(* Logix 5000 project; controller AMANA_DC_PLANT_01 vendor 1 type 14 code 164 rev 31.12; software revision 31.02; part 2 of 9 *)

TYPE Keyence_2_Barcode :
STRUCT
   Trigger_Timer : TIMER;
   Barcode_SRTrigger : BOOL;
   Barcode_ReadIsSuccess : BOOL;
   Barcode_Raw : STRING;
   Barcode_Comma_Position : INT;
   Barcode_1_Length : INT;
   Barcode_2_Length : INT;
   Barcode_2_Start : INT;
   PlaceHolder_ConveyorRunning : BOOL;
   Barcode_1_String : STRING;
   Barcode_2_String : STRING;
   Scanner_Name : STRING;
   Barcode_SRReaderReady : BOOL;
   OneShot : BOOL;
END_STRUCT
END_TYPE

TYPE STRING_12 :
STRUCT
   LEN : DINT;
   DATA : SINT[12];
END_STRUCT
END_TYPE

TYPE STRING_16 :
STRUCT
   LEN : DINT;
   DATA : SINT[16];
END_STRUCT
END_TYPE

TYPE STRING_24 :
STRUCT
   LEN : DINT;
   DATA : SINT[24];
END_STRUCT
END_TYPE

TYPE STRING_4 :
STRUCT
   LEN : DINT;
   DATA : SINT[4];
END_STRUCT
END_TYPE

TYPE STRING_40 :
STRUCT
   LEN : DINT;
   DATA : SINT[40];
END_STRUCT
END_TYPE

TYPE UDT_Current_Status :
STRUCT
   Area : STRING_12;
   Line : STRING_12;
   Shift : DINT;
   _1st_Shift_Avail : BOOL;
   _1st_Shift_Active : BOOL;
   _1st_Shift_Scheduled : BOOL;
   _2nd_Shift_Avail : BOOL;
   _2nd_Shift_Active : BOOL;
   _2nd_Shift_Scheduled : BOOL;
   _3rd_Shift_Avail : BOOL;
   _3rd_Shift_Active : BOOL;
   _3rd_Shift_Scheduled : BOOL;
   DayOfWeek : STRING_16;
   DayOfWeek_Int : DINT;
   Start_Time : STRING_16;
   End_Time : STRING_16;
   _1st_Break_Time : STRING_16;
   _1st_Break_Trigger : BOOL;
   _1st_Break_Active : BOOL;
   _1st_Break_Used : BOOL;
   Lunch_Time : STRING_16;
   Lunch_Trigger : BOOL;
   Lunch_Active : BOOL;
   Lunch_Used : BOOL;
   _2nd_Break_Time : STRING_16;
   _2nd_Break_Trigger : BOOL;
   _2nd_Break_Active : BOOL;
   _2nd_Break_Used : BOOL;
   Rotate_Active : BOOL;
   Rotate_Cmd : BOOL;   // 30 Second Downtime Event to Rotate the Crew
   Scheduled_Units : DINT;
   Line_Rate : DINT;   // Seconds to Construct a Component
   Line_Rate_SP : REAL;
   Units_Remaining : DINT;
   Units_Produced : DINT;
   Units_Scrapped : DINT;
   Units_Lossed : DINT;
   AY_Percent : REAL;
   Shift_Minutes_Remainng : DINT;
   Shift_Seconds_Remaining : DINT;
   DownTime_Code : DINT;
   Flex_Cmd : BOOL;
   Flex_Active : BOOL;
   FlexTo_Line : STRING_16;
   Flex_EndCmd : BOOL;
   Rotate_LEN : REAL;   // seconds
   Brk_LEN : REAL;   // minutes
   Lunch_LEN : REAL;   // minutes
   Break_Stop_On : BOOL;
   Break_Stop_Allowed : BOOL;
   Flex_Stop_On : BOOL;
   Flex_Stop_Allowed : BOOL;
   Rotate_Stop_On : BOOL;
   Rotate_Stop_Allowed : BOOL;
   S1_Scheduled : DINT;
   S2_Scheduled : DINT;
   S3_Scheduled : DINT;
   Shift_Scheduled : BOOL;
   Shift_Active : BOOL;
   RateToMakeSchedule : REAL;
   Theoretical_Units : DINT;
   Standard_LineRate : REAL;
   Running : BOOL;
   State : DINT;
   LineWide_Event : DINT;
END_STRUCT
END_TYPE

TYPE UDT_Daily_Schedule :
STRUCT
   _1st_Shift_Avail : BOOL;
   _1st_Shift_Start : STRING_16;
   _1st_Shift_End : STRING_16;
   _1st_Shift_Break1_Start : STRING_16;
   _1st_Shift_Break1_Length : DINT;   // Minutes
   _1st_Shift_Lunch_Start : STRING_16;
   _1st_Shift_Lunch_Length : DINT;   // Minutes
   _1st_Shift_Break2_Start : STRING_16;
   _1st_Shift_Break2_Length : DINT;   // Minutes
   _2nd_Shift_Avail : BOOL;
   _2nd_Shift_Start : STRING_16;
   _2nd_Shift_End : STRING_16;
   _2nd_Shift_Break1_Start : STRING_16;
   _2nd_Shift_Break1_Length : DINT;   // Minutes
   _2nd_Shift_Lunch_Start : STRING_16;
   _2nd_Shift_Lunch_Length : DINT;   // Minutes
   _2nd_Shift_Break2_Start : STRING_16;
   _2nd_Shift_Break2_Length : DINT;   // Minutes
   _3rd_Shift_Avail : BOOL;
   _3rd_Shift_Start : STRING_16;
   _3rd_Shift_End : STRING_16;
   _3rd_Shift_Break1_Start : STRING_16;
   _3rd_Shift_Break1_Length : DINT;   // Minutes
   _3rd_Shift_Lunch_Start : STRING_16;
   _3rd_Shift_Lunch_Length : DINT;   // Minutes
   _3rd_Shift_Break2_Start : STRING_16;
   _3rd_Shift_Break2_Length : DINT;   // Minutes
   Rotate_Length : DINT;   // Seconds
   Break_Stop_On : BOOL;
   Break_Stop_Allowed : BOOL;
   Flex_Stop_On : BOOL;
   Flex_Stop_Allowed : BOOL;
   Rotate_Stop_On : BOOL;
   Rotate_Stop_Allowed : BOOL;
   S1_Scheduled : DINT;
   S2_Scheduled : DINT;
   S3_Scheduled : DINT;
   RateToMakeSchedule : REAL;
END_STRUCT
END_TYPE

TYPE UDT_ShiftString_Breakdown :
STRUCT
   s1StartHour : STRING_4;
   s1StartMin : STRING_4;
   s1EndHour : STRING_4;
   s1_EndMin : STRING_4;
   s2StartHour : STRING_4;
   s2StartMin : STRING_4;
   s2EndHour : STRING_4;
   s2EndMin : STRING_4;
   s3StartHour : STRING_4;
   s3StartMin : STRING_4;
   s3EndHour : STRING_4;
   s3EndMin : STRING_4;
   break1StartHour : STRING_4;
   break1StartMin : STRING_4;
   break2StartHour : STRING_4;
   break2StartMin : STRING_4;
   lunchStartHour : STRING_4;
   lunchStartMin : STRING_4;
END_STRUCT
END_TYPE

TYPE UDT_SN_Model :
STRUCT
   writeIndex : DINT;
   readIndex : DINT;
   LastReadCode : DINT;
   Serial : STRING_16;
   Model : STRING_16;
   DateTime : STRING_24;
   newData : BOOL;
END_STRUCT
END_TYPE

TYPE UDT_Weekly_Schedule :
STRUCT
   Monday : UDT_Daily_Schedule;
   Tuesday : UDT_Daily_Schedule;
   Wednesday : UDT_Daily_Schedule;
   Thursday : UDT_Daily_Schedule;
   Friday : UDT_Daily_Schedule;
   Saturday : UDT_Daily_Schedule;
   Sunday : UDT_Daily_Schedule;
END_STRUCT
END_TYPE

VAR_GLOBAL   (* controller tags *)
   ay : REAL := 0.84177995;
   DC1_clock_sync : DINT[10] := ([0] := 1998, [1] := 5, [2] := 19, [3] := 23, [4] := 1, [5] := 17);
   DC1_OPCFault : BOOL := 1;
   DC1_to_LN00_Messages : DINT[20] := ([2] := 1, [3] := 1948, [5] := 7, [6] := 5, [7] := 15, [8] := 28, [9] := 15, [10] := 35, [11] := 23, [12] := 58, [14] := 5, [15] := 6, [16] := 58, [17] := 33900, [19] := 1);
        [10]   // CURRENT SCHEDULE SHIFT 2 START MINUTE
        [11]   // CURRENT SCHEDULE SHIFT 2 END HOUR
        [12]   // CURRENT SCHEDULE SHIFT 2 END MINUTE
        [13]   // CURRENT SCHEDULE SHIFT 3 START HOUR
        [14]   // CURRENT SCHEDULE SHIFT 3 START MINUTE
        [15]   // CURRENT SCHEDULE SHIFT 3 END HOUR
        [16]   // CURRENT SCHEDULE SHIFT 3 END MINUTE
        [17]   // CURRENT SCHEDULE AVAILABLE SECONDS
        [19].0   // SHIFT SCHEDULED
        [19].1   // OPC COMMS OKAY
        [2]   // ACTIVE SHIFT
        [3]   // SCHEDULED UNITS
        [5]   // CURRENT SCHEDULE SHIFT 1 START HOUR
        [6]   // CURRENT SCHEDULE SHIFT 1 START MINUTE
        [7]   // CURRENT SCHEDULE SHIFT 1 END HOUR
        [8]   // CURRENT SCHEDULE SHIFT 1 END MINUTE
        [9]   // CURRENT SCHEDULE SHIFT 2 START HOUR
   DC1_to_LN00_Time_sync_Out : MESSAGE;
        MessageParameters(ServiceCode := 16#004d, LocalElement := DC1_clock_sync[0], ...)
   fifi_unload : DINT;
   LN00_1st_Station_Break_Code : DINT := 16;
   LN00_COUNTS_FROM_IGN_DB : DINT := 291;
   LN00_COUNTS_FROM_IGN_DB_msg : MESSAGE;
        MessageParameters(ServiceCode := 16#004d, LocalElement := LN00_COUNTS_FROM_IGN_DB, ...)
   LN00_FPY : REAL := 67.69;
   LN00_MainLine_MSG_Out : MESSAGE;
        MessageParameters(ServiceCode := 16#004d, LocalElement := DC1_to_LN00_Messages[0], ...)
   LN00_MLC_Downtime : BOOL;
   LN00_Schedule : UDT_Current_Status := (Line := 'LN00', Shift := 1, _1st_Shift_Avail := 1, _1st_Shift_Active := 1, _1st_Shift_Scheduled := 1, _2nd_Shift_Scheduled := 1, _3rd_Shift_Scheduled := 1, DayOfWeek := 'Mon', DayOfWeek_Int := 1, Start_Time := '07:05', End_Time := '15:28', _1st_Break_Time := '09:10', Lunch_Time := '12:10', _2nd_Break_Time := '20:30', Scheduled_Units := 1948, Line_Rate := 34, Units_Remaining := 1267, Units_Produced := 681, Units_Lossed := 128, AY_Percent := 84.17799, Break_Stop_On := 1, Break_Stop_Allowed := 1, Shift_Scheduled := 1, Shift_Active := 1, Theoretical_Units := 809, State := 5, LineWide_Event := 16);
   LN00_ScheduleUnits_Produced_from_line : DINT := 338;
   LN00_SNModel_Array : UDT_SN_Model[50] := ([0].LastReadCode := 1, [0].Serial := 'M91940581', [0].Model := 'WED4815EW1', [0].DateTime := '5/10/2019 17:12:14', [1].readIndex := 1, [1].LastReadCode := 1, [1].Serial := 'M91940582', [1].Model := 'WED4815EW1', [1].DateTime := '5/10/2019 17:12:25', [2].readIndex := 2, [2].LastReadCode := -1, [2].Serial := 'M91940583', [2].Model := 'WED4815EW1', [2].DateTime := '5/10/2019 17:12:37', [3].readIndex := 3, [3].LastReadCode := 1, [3].Serial := 'M91940584', [3].Model := 'WED4815EW1', [3].DateTime := '5/10/2019 17:12:48', [4].readIndex := 4, [4].LastReadCode := 1, [4].Serial := 'M91940585', [4].Model := 'WED4815EW1', [4].DateTime := '5/10/2019 17:13:00', [5].readIndex := 5, [5].LastReadCode := 1, [5].Serial := 'M91940586', [5].Model := 'WED4815EW1', [5].DateTime := '5/10/2019 17:13:11', [6].readIndex := 6, [6].LastReadCode := 1, [6].Serial := 'M91940587', [6].Model := 'WED4815EW1', [6].DateTime := '5/10/2019 17:13:22', [7].readIndex := 7, [7].LastReadCode := 1, [7].Serial := 'M91940588', [7].Model := 'WED4815EW1', [7].DateTime := '5/10/2019 17:13:34', [8].readIndex := 8, [8].LastReadCode := 1, [8].Serial := 'M91940589', [8].Model := 'WED4815EW1', [8].DateTime := '5/10/2019 17:13:46', [9].readIndex := 9, [9].LastReadCode := 1, [9].Serial := 'M91940590', [9].Model := 'WED4815EW1', [9].DateTime := '5/10/2019 17:13:57', [10].readIndex := 10, [10].LastReadCode := 1, [10].Serial := 'M91940591', [10].Model := 'WED4815EW1', [10].DateTime := '5/10/2019 17:14:09', [11].readIndex := 11, [11].LastReadCode := 1, [11].Serial := 'M91940592', [11].Model := 'WED4815EW1', [11].DateTime := '5/10/2019 17:14:20', [12].readIndex := 12,
        [12].LastReadCode := 1, [12].Serial := 'M91940593', [12].Model := 'WED4815EW1', [12].DateTime := '5/10/2019 17:14:32', [13].readIndex := 13, [13].LastReadCode := 1, [13].Serial := 'M91940594', [13].Model := 'WED4815EW1', [13].DateTime := '5/10/2019 17:14:43', [14].readIndex := 14, [14].LastReadCode := 1, [14].Serial := 'M91940595', [14].Model := 'WED4815EW1', [14].DateTime := '5/10/2019 17:14:55', [15].readIndex := 15, [15].LastReadCode := 1, [15].Serial := 'M91940596', [15].Model := 'WED4815EW1', [15].DateTime := '5/10/2019 17:15:06', [16].readIndex := 16, [16].LastReadCode := 1, [16].Serial := 'M91940597', [16].Model := 'WED4815EW1', [16].DateTime := '5/10/2019 17:15:17', [17].readIndex := 17, [17].LastReadCode := 1, [17].Serial := 'M91940598', [17].Model := 'WED4815EW1', [17].DateTime := '5/10/2019 17:15:29', [18].readIndex := 18, [18].LastReadCode := 1, [18].Serial := 'M91940599', [18].Model := 'WED4815EW1', [18].DateTime := '5/10/2019 17:15:40', [19].readIndex := 19, [19].LastReadCode := 1, [19].Serial := 'M91940599$00$00$00$00$00$00$00', [19].Model := 'WED4815EW1', [19].DateTime := '5/10/2019 17:15:43', [20].readIndex := 20, [20].LastReadCode := -2, [20].Model := 'WED4815EW1', [20].DateTime := '5/10/2019 17:15:52', [21].readIndex := 21, [21].LastReadCode := -2, [21].Serial := 'M91940600', [21].Model := 'WED4815EW1', [21].DateTime := '5/10/2019 17:16:03', [22].readIndex := 22, [22].LastReadCode := 1, [22].Serial := 'M91940601', [22].Model := 'WED4815EW1', [22].DateTime := '5/10/2019 17:16:06', [23].readIndex := 23, [23].LastReadCode := 1, [23].Model := 'WED4815EW1', [23].DateTime := '5/10/2019 17:16:13', [24].readIndex := 24, [24].LastReadCode := -2, [24].Serial := 'M91940602',
        [24].Model := 'WED4815EW1', [24].DateTime := '5/10/2019 17:16:15', [25].readIndex := 25, [25].LastReadCode := 1, [25].Serial := 'M91940603', [25].Model := 'WED4815EW1', [25].DateTime := '5/10/2019 17:16:38', [26].readIndex := 26, [26].LastReadCode := 1, [26].Serial := 'M91940604', [26].Model := 'WED4815EW1', [26].DateTime := '5/10/2019 17:16:49', [27].readIndex := 27, [27].LastReadCode := 1, [27].Serial := 'M91940605', [27].Model := 'WED4815EW1', [27].DateTime := '5/10/2019 17:17:01', [28].readIndex := 28, [28].LastReadCode := 1, [28].Serial := 'M91940606', [28].Model := 'WED4815EW1', [28].DateTime := '5/10/2019 17:17:11', [29].readIndex := 29, [29].LastReadCode := 1, [29].Serial := 'M91940607', [29].Model := 'WED4815EW1', [29].DateTime := '5/10/2019 17:17:23', [30].readIndex := 30, [30].LastReadCode := 1, [30].Serial := 'M91940608', [30].Model := 'WED4815EW1', [30].DateTime := '5/10/2019 17:17:35', [31].readIndex := 31, [31].LastReadCode := 1, [31].Serial := 'M91940609', [31].Model := 'WED4815EW1', [31].DateTime := '5/10/2019 17:17:46', [32].readIndex := 32, [32].LastReadCode := 1, [32].Serial := 'M91940610', [32].Model := 'WED4815EW1', [32].DateTime := '5/10/2019 17:17:58', [33].readIndex := 33, [33].LastReadCode := -2, [33].Serial := 'M91940611', [33].Model := 'WED4815EW1', [33].DateTime := '5/10/2019 17:18:09', [34].readIndex := 34, [34].LastReadCode := 1, [34].Serial := 'M91940565', [34].Model := 'WED4815EW1', [34].DateTime := '5/10/2019 17:09:11', [35].readIndex := 35, [35].LastReadCode := 1, [35].Serial := 'M91940566', [35].Model := 'WED4815EW1', [35].DateTime := '5/10/2019 17:09:22', [36].readIndex := 36, [36].LastReadCode := 1, [36].Serial := 'M91940567',
        [36].Model := 'WED4815EW1', [36].DateTime := '5/10/2019 17:09:34', [37].readIndex := 37, [37].LastReadCode := 1, [37].Serial := 'M91940568', [37].Model := 'WED4815EW1', [37].DateTime := '5/10/2019 17:09:45', [38].readIndex := 38, [38].LastReadCode := 1, [38].Serial := 'M91940569', [38].Model := 'WED4815EW1', [38].DateTime := '5/10/2019 17:09:57', [39].readIndex := 39, [39].LastReadCode := 1, [39].Serial := 'M91940570', [39].Model := 'WED4815EW1', [39].DateTime := '5/10/2019 17:10:08', [40].readIndex := 40, [40].LastReadCode := 1, [40].Serial := 'M91940571', [40].Model := 'WED4815EW1', [40].DateTime := '5/10/2019 17:10:19', [41].readIndex := 41, [41].LastReadCode := 1, [41].Serial := 'M91940572', [41].Model := 'WED4815EW1', [41].DateTime := '5/10/2019 17:10:31', [42].readIndex := 42, [42].LastReadCode := 1, [42].Serial := 'M91940573', [42].Model := 'WED4815EW1', [42].DateTime := '5/10/2019 17:10:43', [43].readIndex := 43, [43].LastReadCode := 1, [43].Serial := 'M91940574', [43].Model := 'WED4815EW1', [43].DateTime := '5/10/2019 17:10:54', [44].readIndex := 44, [44].LastReadCode := 1, [44].Serial := 'M91940575', [44].Model := 'WED4815EW1', [44].DateTime := '5/10/2019 17:11:05', [45].readIndex := 45, [45].LastReadCode := 1, [45].Serial := 'M91940576', [45].Model := 'WED4815EW1', [45].DateTime := '5/10/2019 17:11:16', [46].readIndex := 46, [46].LastReadCode := 1, [46].Serial := 'M91940577', [46].Model := 'WED4815EW1', [46].DateTime := '5/10/2019 17:11:28', [47].readIndex := 47, [47].LastReadCode := 1, [47].Serial := 'M91940578', [47].Model := 'WED4815EW1', [47].DateTime := '5/10/2019 17:11:40', [48].readIndex := 48, [48].LastReadCode := 1, [48].Serial := 'M91940579',
        [48].Model := 'WED4815EW1', [48].DateTime := '5/10/2019 17:11:51', [49].readIndex := 49, [49].LastReadCode := 1, [49].Serial := 'M91940580', [49].Model := 'WED4815EW1', [49].DateTime := '5/10/2019 17:12:03');
   LN00_SNModel_CurrentRead : UDT_SN_Model := (writeIndex := 33, Serial := 'M91940581', Model := 'WED4815EW1', DateTime := '5/10/2019 17:12:14');
   LN00_SNModel_MSG : MESSAGE;
        MessageParameters(ServiceCode := 16#004c, LocalElement := LN00_SNModel_STR[0], ...)
   LN00_SNModel_STR : STRING[10] := ([0] := 'M91940611', [1] := 'WED4815EW1', [2] := '5/10/2019 17:18:12');
   LN00_to_DC1_Main_Messages_0 : DINT[40] := ([4] := 681, [5] := 7812, [6] := 34, [9] := 2, [15] := 6769, [18] := 809, [19] := 142, [39] := 126); {produced}
   LN00_to_DC1_Main_Messages_1 : DINT[120] := ([2] := 900, [7] := 900, [8] := 900, [9] := 900, [10] := 900);
   LN00_to_DC1_Main_Messages_2 : DINT[120];
   LN00_to_DC1_Main_Messages_3 : DINT[120];
   LN00_to_DC1_Main_Messages_4 : DINT[120];
   LN00_to_DC1_Main_Messages_5 : DINT[120];
   LN00_to_DC1_Main_Messages_6 : DINT[120];
   LN00_to_DC1_Main_MSG1 : MESSAGE;
        MessageParameters(ServiceCode := 16#004c, LocalElement := LN00_to_DC1_Main_Messages_1[1], ...)
   LN00_to_DC1_Main_MSG2 : MESSAGE;
        MessageParameters(ServiceCode := 16#004c, LocalElement := LN00_to_DC1_Main_Messages_2[1], ...)
   LN00_to_DC1_Main_MSG3 : MESSAGE;
   LN00_to_DC1_Main_MSG4 : MESSAGE;
   LN00_to_DC1_Main_MSG5 : MESSAGE;
   LN00_to_DC1_Main_MSG6 : MESSAGE;
        MessageParameters(ServiceCode := 16#004c, LocalElement := LN00_to_DC1_Main_Messages_3[11], ...)
   LN00_Toggle_CountSource : BOOL;
   LN00_Weekly_Schedule : UDT_Weekly_Schedule := (Monday._1st_Shift_Avail := 1, Monday._1st_Shift_Start := '07:05', Monday._1st_Shift_End := '15:28', Monday._1st_Shift_Break1_Start := '09:10', Monday._1st_Shift_Break1_Length := 15, Monday._1st_Shift_Lunch_Start := '12:10', Monday._1st_Shift_Lunch_Length := 30, Monday._1st_Shift_Break2_Start := '20:30', Monday._1st_Shift_Break2_Length := 15, Monday._2nd_Shift_Avail := 1, Monday._2nd_Shift_Start := '15:35', Monday._2nd_Shift_End := '23:58', Monday._2nd_Shift_Break1_Start := '17:45', Monday._2nd_Shift_Break1_Length := 15, Monday._2nd_Shift_Lunch_Start := '20:30', Monday._2nd_Shift_Lunch_Length := 30, Monday._2nd_Shift_Break2_Start := '12:10', Monday._2nd_Shift_Break2_Length := 15, Monday._3rd_Shift_Avail := 1, Monday._3rd_Shift_Start := '00:05', Monday._3rd_Shift_End := '06:58', Monday._3rd_Shift_Break1_Start := '01:00', Monday._3rd_Shift_Break1_Length := 15, Monday._3rd_Shift_Lunch_Start := '03:00', Monday._3rd_Shift_Lunch_Length := 30, Monday._3rd_Shift_Break2_Start := '04:00', Monday._3rd_Shift_Break2_Length := 15, Monday.S1_Scheduled := 1948, Monday.S2_Scheduled := 1948, Monday.S3_Scheduled := 507, Tuesday._1st_Shift_Avail := 1, Tuesday._1st_Shift_Start := '07:05', Tuesday._1st_Shift_End := '15:28', Tuesday._1st_Shift_Break1_Start := '09:10', Tuesday._1st_Shift_Break1_Length := 15, Tuesday._1st_Shift_Lunch_Start := '12:10', Tuesday._1st_Shift_Lunch_Length := 30, Tuesday._1st_Shift_Break2_Start := '20:30', Tuesday._1st_Shift_Break2_Length := 15, Tuesday._2nd_Shift_Avail := 1, Tuesday._2nd_Shift_Start := '15:35', Tuesday._2nd_Shift_End := '23:58', Tuesday._2nd_Shift_Break1_Start := '17:45', Tuesday._2nd_Shift_Break1_Length := 15, Tuesday._2nd_Shift_Lunch_Start := '20:30', Tuesday._2nd_Shift_Lunch_Length := 30, Tuesday._2nd_Shift_Break2_Start := '12:10', Tuesday._2nd_Shift_Break2_Length := 15, Tuesday._3rd_Shift_Avail := 1, Tuesday._3rd_Shift_Start := '00:05', Tuesday._3rd_Shift_End := '06:58', Tuesday._3rd_Shift_Break1_Start := '01:00', Tuesday._3rd_Shift_Break1_Length := 15, Tuesday._3rd_Shift_Lunch_Start := '03:00', Tuesday._3rd_Shift_Lunch_Length := 30, Tuesday._3rd_Shift_Break2_Start := '04:00', Tuesday._3rd_Shift_Break2_Length := 15, Tuesday.S1_Scheduled := 1948, Tuesday.S2_Scheduled := 1948, Tuesday.S3_Scheduled := 507,
        Wednesday._1st_Shift_Avail := 1, Wednesday._1st_Shift_Start := '07:05', Wednesday._1st_Shift_End := '15:28', Wednesday._1st_Shift_Break1_Start := '09:10', Wednesday._1st_Shift_Break1_Length := 15, Wednesday._1st_Shift_Lunch_Start := '12:10', Wednesday._1st_Shift_Lunch_Length := 30, Wednesday._1st_Shift_Break2_Start := '20:30', Wednesday._1st_Shift_Break2_Length := 15, Wednesday._2nd_Shift_Avail := 1, Wednesday._2nd_Shift_Start := '15:35', Wednesday._2nd_Shift_End := '23:58', Wednesday._2nd_Shift_Break1_Start := '17:45', Wednesday._2nd_Shift_Break1_Length := 15, Wednesday._2nd_Shift_Lunch_Start := '20:30', Wednesday._2nd_Shift_Lunch_Length := 30, Wednesday._2nd_Shift_Break2_Start := '12:10', Wednesday._2nd_Shift_Break2_Length := 15, Wednesday._3rd_Shift_Avail := 1, Wednesday._3rd_Shift_Start := '00:05', Wednesday._3rd_Shift_End := '06:58', Wednesday._3rd_Shift_Break1_Start := '01:00', Wednesday._3rd_Shift_Break1_Length := 15, Wednesday._3rd_Shift_Lunch_Start := '03:00', Wednesday._3rd_Shift_Lunch_Length := 30, Wednesday._3rd_Shift_Break2_Start := '04:00', Wednesday._3rd_Shift_Break2_Length := 15, Wednesday.S1_Scheduled := 1948, Wednesday.S2_Scheduled := 1948, Wednesday.S3_Scheduled := 507, Thursday._1st_Shift_Avail := 1, Thursday._1st_Shift_Start := '07:05', Thursday._1st_Shift_End := '15:28', Thursday._1st_Shift_Break1_Start := '09:10', Thursday._1st_Shift_Break1_Length := 15, Thursday._1st_Shift_Lunch_Start := '12:10', Thursday._1st_Shift_Lunch_Length := 30, Thursday._1st_Shift_Break2_Start := '20:30', Thursday._1st_Shift_Break2_Length := 15, Thursday._2nd_Shift_Avail := 1, Thursday._2nd_Shift_Start := '15:35', Thursday._2nd_Shift_End := '23:58', Thursday._2nd_Shift_Break1_Start := '17:45', Thursday._2nd_Shift_Break1_Length := 15, Thursday._2nd_Shift_Lunch_Start := '20:30', Thursday._2nd_Shift_Lunch_Length := 30, Thursday._2nd_Shift_Break2_Start := '12:10', Thursday._2nd_Shift_Break2_Length := 15, Thursday._3rd_Shift_Avail := 1, Thursday._3rd_Shift_Start := '00:05', Thursday._3rd_Shift_End := '06:58', Thursday._3rd_Shift_Break1_Start := '01:00', Thursday._3rd_Shift_Break1_Length := 15, Thursday._3rd_Shift_Lunch_Start := '03:00', Thursday._3rd_Shift_Lunch_Length := 30, Thursday._3rd_Shift_Break2_Start := '04:00', Thursday._3rd_Shift_Break2_Length := 15, Thursday.S1_Scheduled := 1948, Thursday.S2_Scheduled := 1948, Thursday.S3_Scheduled := 507,
        Friday._1st_Shift_Avail := 1, Friday._1st_Shift_Start := '07:05', Friday._1st_Shift_End := '15:28', Friday._1st_Shift_Break1_Start := '09:10', Friday._1st_Shift_Break1_Length := 15, Friday._1st_Shift_Lunch_Start := '12:10', Friday._1st_Shift_Lunch_Length := 30, Friday._1st_Shift_Break2_Start := '20:30', Friday._1st_Shift_Break2_Length := 15, Friday._2nd_Shift_Avail := 1, Friday._2nd_Shift_Start := '15:35', Friday._2nd_Shift_End := '23:58', Friday._2nd_Shift_Break1_Start := '17:45', Friday._2nd_Shift_Break1_Length := 15, Friday._2nd_Shift_Lunch_Start := '20:30', Friday._2nd_Shift_Lunch_Length := 30, Friday._2nd_Shift_Break2_Start := '12:10', Friday._2nd_Shift_Break2_Length := 15, Friday._3rd_Shift_Avail := 1, Friday._3rd_Shift_Start := '00:05', Friday._3rd_Shift_End := '06:58', Friday._3rd_Shift_Break1_Start := '01:00', Friday._3rd_Shift_Break1_Length := 15, Friday._3rd_Shift_Lunch_Start := '03:00', Friday._3rd_Shift_Lunch_Length := 30, Friday._3rd_Shift_Break2_Start := '04:00', Friday._3rd_Shift_Break2_Length := 15, Friday.S1_Scheduled := 1948, Friday.S2_Scheduled := 1948, Friday.S3_Scheduled := 507, Saturday._1st_Shift_Start := '07:05', Saturday._1st_Shift_End := '15:28', Saturday._1st_Shift_Break1_Start := '09:10', Saturday._1st_Shift_Break1_Length := 15, Saturday._1st_Shift_Lunch_Start := '12:10', Saturday._1st_Shift_Lunch_Length := 30, Saturday._1st_Shift_Break2_Start := '18:45', Saturday._1st_Shift_Break2_Length := 15, Saturday._2nd_Shift_Start := '15:35', Saturday._2nd_Shift_End := '23:58', Saturday._2nd_Shift_Break1_Start := '17:45', Saturday._2nd_Shift_Break1_Length := 15, Saturday._2nd_Shift_Lunch_Start := '20:30', Saturday._2nd_Shift_Lunch_Length := 30, Saturday._2nd_Shift_Break2_Start := '12:10', Saturday._2nd_Shift_Break2_Length := 15, Saturday._3rd_Shift_Start := '00:05', Saturday._3rd_Shift_End := '06:58', Saturday._3rd_Shift_Break1_Start := '01:00', Saturday._3rd_Shift_Break1_Length := 15, Saturday._3rd_Shift_Lunch_Start := '03:00', Saturday._3rd_Shift_Lunch_Length := 30, Saturday._3rd_Shift_Break2_Start := '05:00', Saturday._3rd_Shift_Break2_Length := 15, Sunday._1st_Shift_Start := '07:05', Sunday._1st_Shift_End := '15:28', Sunday._1st_Shift_Break1_Start := '09:10', Sunday._1st_Shift_Break1_Length := 15, Sunday._1st_Shift_Lunch_Start := '12:10', Sunday._1st_Shift_Lunch_Length := 30,
        Sunday._1st_Shift_Break2_Start := '18:45', Sunday._1st_Shift_Break2_Length := 15, Sunday._2nd_Shift_Start := '15:35', Sunday._2nd_Shift_End := '23:58', Sunday._2nd_Shift_Break1_Start := '17:45', Sunday._2nd_Shift_Break1_Length := 15, Sunday._2nd_Shift_Lunch_Start := '20:30', Sunday._2nd_Shift_Lunch_Length := 30, Sunday._2nd_Shift_Break2_Start := '12:10', Sunday._2nd_Shift_Break2_Length := 15, Sunday._3rd_Shift_Start := '00:05', Sunday._3rd_Shift_End := '06:58', Sunday._3rd_Shift_Break1_Start := '01:00', Sunday._3rd_Shift_Break1_Length := 140, Sunday._3rd_Shift_Lunch_Start := '03:00', Sunday._3rd_Shift_Lunch_Length := 30, Sunday._3rd_Shift_Break2_Start := '05:00', Sunday._3rd_Shift_Break2_Length := 10);
   LN00DAM01 : DINT;
   LN00DAM02 : DINT;
   LN00DAM03 : DINT;
   LN00DAM04 : DINT;
   LN00DAM05 : DINT;
   LN00DAM06 : DINT;
   LN00DAM07 : DINT;
   LN00DAM08 : DINT;
   LN00DAM09 : DINT;
   LN00DBM02 : DINT;
   LN00DBM03 : DINT;
   LN00DCM04 : DINT;
   LN00DCM05 : DINT;
   LN00DCM06 : DINT;
   LN00DCM07 : DINT;
   LN00DCM08 : DINT;
   LN00DCM09 : DINT;
   LN00DCM10 : DINT;
   LN00DCM11 : DINT;
   LN00DCM12 : DINT;
   LN00DCM13 : DINT;
   LN00DCM14 : DINT;
   LN00DCM15 : DINT;
   LN00DCM16 : DINT;
   LN00DCM17 : DINT;
   LN00DCM18 : DINT;
   LN00DCM19 : DINT;
   LN00DCM20 : DINT;
   LN00DCM21 : DINT;
   LN00DCM22 : DINT;
   LN00DCM23 : DINT;
   LN00DCM24 : DINT;
   LN00DCM25 : DINT;
   LN00DCM26 : DINT;
   LN00DCM27 : DINT;
   LN00DCM28 : DINT;
   LN00DCM29 : DINT;
   LN00DCM30 : DINT;
   LN00DCM31 : DINT;
   LN00DCM32 : DINT;
   LN00DCM33 : DINT;
   LN00DCM34 : DINT;
   LN00DCM35 : DINT;
   LN00DCM36 : DINT;
   LN00DCM37 : DINT;
   LN00DCM38 : DINT;
   LN00DCM39 : DINT;
   LN00DCM40 : DINT;
   LN00DDM01 : DINT;
   LN00DDM02 : DINT;
   LN00DDM03 : DINT;
   LN00DDM04 : DINT;
   LN00DDM05 : DINT;
   LN00DDM06 : DINT;
   LN00DDM07 : DINT;
   LN00DDM08 : DINT;
   LN00DDM09 : DINT;
   LN00DDM10 : DINT;
   LN00DDM11 : DINT;
   LN00DDM12 : DINT;
   LN00DDM13 : DINT;
   LN00DDM14 : DINT;
   LN00DDM15 : DINT;
   LN00DDM16 : DINT;
   LN00DDM17 : DINT;
   LN00DDM18 : DINT;
   LN00DDM19 : DINT;
   LN00DDM20 : DINT;
   LN00DDM21 : DINT;
   LN00DDM22 : DINT;
   LN00DDM23 : DINT;
   LN00DDM24 : DINT;
   LN00DDM25 : DINT;
   LN00DDM26 : DINT;
   LN00DDM27 : DINT;
   LN00DDM28 : DINT;
   LN00DEM01 : DINT;
   LN00DEM02 : DINT;
   LN00DEM03 : DINT;
   LN00DEM04 : DINT;
   LN00DEM05 : DINT;
   LN00DEM06 : DINT;
   LN00DEM07 : DINT;
   LN00DEM08 : DINT;
   LN00DEM09 : DINT;
   LN00DEM10 : DINT;
   LN00DEM11 : DINT;
   LN00DEM12 : DINT;
   LN00DEM13 : DINT;
   LN00DEM14 : DINT;
   LN00DEM15 : DINT;
   LN00DEM16 : DINT;
   LN00DEM17 : DINT;
   LN00DEM18 : DINT;
   LN00DEM19 : DINT;
   LN00DEM20 : DINT;
   LN00DEM21 : DINT;
   LN00DEM22 : DINT;
   LN00DEM23 : DINT;
   LN00DEM24 : DINT;
   LN00DEM25 : DINT;
   LN00DEM26 : DINT;
   LN00DEM27 : DINT;
   LN00DEM28 : DINT;
   LN00DEM29 : DINT;
   LN00DEM30 : DINT;
   LN00DEM31 : DINT;
   LN00DEM32 : DINT;
   LN00DEM33 : DINT;
   LN00DEM34 : DINT;
   LN00DEM35 : DINT;
   LN00DEM36 : DINT;
   LN00DEM37 : DINT;
   LN00DEM38 : DINT;
   LN00DEM39 : DINT;
   LN00DEM40 : DINT;
   LN00DEM41 : DINT;
   LN00DEM42 : DINT;
   LN00DEM43 : DINT;
   LN00DEM44 : DINT;
   LN00DEM45 : DINT;
   LN00DEM46 : DINT;
   LN00DEM47 : DINT;
   LN00DEM48 : DINT;
   LN00DEM49 : DINT;
   LN00DEM50 : DINT;
   LN00DEM51 : DINT;
   LN00DEM52 : DINT;
   LN00DEM53 : DINT;
   LN00DEM54 : DINT;
   LN00DEM55 : DINT;
   LN00DEM56 : DINT;
   LN00DEM57 : DINT;
   LN00DEM58 : DINT;
   LN00DEM59 : DINT;
   LN00DEM60 : DINT;
   LN00DEM61 : DINT;
   LN00DEM62 : DINT;
   LN00DEM63 : DINT;
   LN00DEM64 : DINT;
   LN00DEM65 : DINT;
   LN00DEM66 : DINT;
   LN00DEM67 : DINT;
   LN00DEM68 : DINT;
   LN00DEM69 : DINT;
   LN00DEM70 : DINT;
   LN00DEM71 : DINT;
   LN00DEM72 : DINT;
   LN00DEM73 : DINT;
   LN00DEM74 : DINT;
   LN00DEM75 : DINT;
   LN00DEM76 : DINT;
   LN00DEM77 : DINT;
   LN00DEM78 : DINT;
   LN00DEM79 : DINT;
   LN00DEM80 : DINT;
   LN00DEM81 : DINT;
   LN00DEM82 : DINT;
   LN00DEM83 : DINT;
   LN00DEM84 : DINT;
   LN00DEM85 : DINT;
   LN00DEM86 : DINT;
   LN00DEM87 : DINT;
   LN00DEM88 : DINT;
   LN00DEM89 : DINT;
   LN00DEM90 : DINT;
   LN00DEM91 : DINT;
   LN00DEM92 : DINT;
   LN00DEM93 : DINT;
   LN00DEM94 : DINT;
   LN00DEM95 : DINT;
   LN00DEM96 : DINT;
   LN00DEM97 : DINT;
   LN00DEM98 : DINT;
   LN00DFM01 : DINT;
   LN00DFM02 : DINT;
   LN00DFM03 : DINT;
   LN00DFM04 : DINT;
   LN00DFM05 : DINT;
   LN00DFM06 : DINT;
   LN00DFM07 : DINT;
   LN00DFM08 : DINT;
   LN00DFM09 : DINT;
   LN00DFM10 : DINT;
   LN00DFM11 : DINT;
   LN00DFM12 : DINT;
   LN00DFM13 : DINT;
   LN00DFM14 : DINT;
   LN00DFM15 : DINT;
   LN00DFM16 : DINT;
   LN00DFM17 : DINT;
   LN00DFM18 : DINT;
   LN00DFM19 : DINT;
   LN00DFM20 : DINT;
   LN00DFM21 : DINT;
   LN00DFM22 : DINT;
   LN00DFM23 : DINT;
   LN00DFM24 : DINT;
   LN00DFM25 : DINT;
   LN00DFM26 : DINT;
   LN00DFM27 : DINT;
   LN00DFM28 : DINT;
   LN00DFM29 : DINT;
   LN00DFM30 : DINT;
   LN00DFM31 : DINT;
   LN00DFM32 : DINT;
   LN00DFM33 : DINT;
   LN00DFM34 : DINT;
   LN00DFM35 : DINT;
   LN00EAM00 : DINT := 16;
   LN00EBM00 : DINT;
   LN00EDM00 : DINT;
   msg192_reset_timer : TIMER := (PRE := 3000);
   null : STRING;
   OH_Barcode_Model_CLEARPACK : STRING := 'WRB322DMBM 03';
   OH_Barcode_Model_DOCKSORTING : STRING;
   OH_Barcode_Model_LN4 : STRING;
   OH_Barcode_Model_LN467MERGE : STRING;
   OH_Barcode_Model_LN6 : STRING;
   OH_Barcode_Model_LN67MERGE : STRING;
   OH_Barcode_Model_LN7 : STRING;
   OH_Barcode_Model_LONGTERMEAST : STRING;
   OH_Barcode_Model_LONGTERMWEST : STRING;
   OH_Barcode_Model_WAREHOUSENORTH : STRING;
   OH_Barcode_Model_WAREHOUSESOUTH : STRING;
   OH_Barcode_Serial_CLEARPACK : STRING := 'KC1814086';
   OH_Barcode_Serial_DOCKSORTING : STRING;
   OH_Barcode_Serial_LN4 : STRING;
   OH_Barcode_Serial_LN467MERGE : STRING;
   OH_Barcode_Serial_LN6 : STRING;
   OH_Barcode_Serial_LN67MERGE : STRING;
   OH_Barcode_Serial_LN7 : STRING;
   OH_Barcode_Serial_LONGTERMEAST : STRING;
   OH_Barcode_Serial_LONGTERMWEST : STRING;
   OH_Barcode_Serial_WAREHOUSENORTH : STRING;
   OH_Barcode_Serial_WAREHOUSESOUTH : STRING;
   Previous_Shift_Count : DINT;
   Read_From_Clearpack : INT[16] := ([0] := 1);
        [0].0   // Clearpack P30 Running
   Read_From_Clearpack_1 : MESSAGE;
        MessageParameters(ServiceCode := 16#004c, LocalElement := Read_From_Clearpack[0], ...)
   Read_From_L4_1 : MESSAGE;
   Read_From_L6_1 : MESSAGE;
   Read_From_L7_1 : MESSAGE;
   Read_From_Merge : DINT[8] := ([0] := 1);
   Read_From_Merge_1 : MESSAGE;
        MessageParameters(ServiceCode := 16#004c, LocalElement := Read_From_Merge[0], ...)
   Read_From_Sort_1 : MESSAGE;
   scc : CONTROL := (LEN := 60, POS := 59);   // Shift Count History
   Shift_count_history : DINT[62] := ([22] := 1, [40] := 1, [41] := 1);
   Shift_reset_timer : TIMER := (PRE := 2000);
   THEORETICAL_TEST : BOOL := 1;
END_VAR

PROGRAM LN00   (* main routine MainRoutine *)
VAR
   Average_Array : DINT[20] := ([0] := 30000, [1] := 24250, [2] := 30000, [3] := 30000, [4] := 30000, [5] := 30000, [6] := 30000, [7] := 30000, [8] := 30000, [9] := 30000);   // AVERAGE UNIT ASSEMBLY TIME (LAST 10 UNITS)
   Average_Sum : DINT := 294250;
   Averaged_LineSpeed : REAL := 29.425;
   badModel : STRING_40;
   Break1_Hour : DINT := 9;
   Break1_Hour_String : STRING_4 := '09';
   Break1_Length : DINT := 15;
   Break1_MilliRemain : DINT := 540000;
   Break1_Min : DINT := 10;
   Break1_Min_String : STRING_4 := '10';
   Break1_MinDisplay : DINT;
   Break1_SecDisplay : DINT;
   Break1_SecRemain : DINT := 540;
   Break1_SecWholeMin : DINT := 540;
   Break1_Timer : TIMER := (PRE := 540000);
   Break2_Hour : DINT := 20;
   Break2_Hour_String : STRING_4 := '20';
   Break2_Length : DINT := 15;
   Break2_MilliRemain : DINT := 540000;
   Break2_Min : DINT := 30;
   Break2_Min_String : STRING_4 := '30';
   Break2_MinDisplay : DINT := 9;
   Break2_SecDisplay : DINT;
   Break2_SecRemain : DINT := 540;
   Break2_SecWholeMin : DINT := 540;
   Break2_Timer : TIMER := (PRE := 540000);
   Break_1stStation : BOOL := 1;
   Break_Group1 : BOOL;
   Break_Group2 : BOOL;
   Break_Group3 : BOOL;
   Break_Group4 : BOOL;
   Break_Group5 : BOOL;
   Break_Group6 : BOOL;
   Break_LineWide : BOOL := 1;
   Break_WorkCenter : BOOL := 1;
   Break_Workstation : BOOL := 1;
   CurrentSchedule : UDT_ShiftString_Breakdown := (s1StartHour := '07', s1StartMin := '05', s1EndHour := '15', s1_EndMin := '28', s2StartHour := '15', s2StartMin := '35', s2EndHour := '23', s2EndMin := '58', s3StartHour := '00', s3StartMin := '05', s3EndHour := '06', s3EndMin := '58');
   End_Hour : DINT := 15;
   End_Hour_String : STRING_4 := '15';
   End_Min : DINT := 28;
   End_Min_String : STRING_4 := '28';
   firstCharacter : STRING_40 := 'W';
   FlexTimer_HoursDisplay : DINT;
   FlexTimer_MinutesDisplay : DINT;
   FlexTimer_SecondsDisplay : DINT;
   FlexTimertoHours : DINT;
   FlexTimertoMinutes : DINT;
   FlexTimertoSeconds : DINT;
   HoursFromMidnight : DINT;
   HoursFromMidnight_Remain : DINT := -17;
   HoursTilMidnight : DINT := 9;
   HoursTilMidnight_Remain : DINT;
   LineRate_perSecond_scheduled : REAL := 0.087789856;
   LN06_Flex_Timer : TIMER := (PRE := 28800000);
   LN06_Rotate_Timer : TIMER;
   Local_Timer : TIMER[10] := ([0].PRE := 30000, [1].PRE := 4000, [2].PRE := 8000, [3].PRE := 2000, [3].ACC := 1935, [3].EN := 1, [3].TT := 1, [4].PRE := 280, [4].ACC := 176, [4].EN := 1, [4].TT := 1);
        [0]   // UNIT ASSEMBLY TIMER
        [1]   // BARCODE TRANSFER TO LODESTAR TRIGGER TIMER
        [2]   // BARCOE TRANFER TO LODESTAR SECOND CHANCE TIMER
        [3]   // LINE PLC WRITE MESSAGE INSTRUCTION TIMER
        [4]   // LINE PLC READ MESSAGE INSTRUCTION TIMER
   Lunch_Hour : DINT := 12;
   Lunch_Hour_String : STRING_4 := '12';
   Lunch_Length : DINT := 30;
   Lunch_MilliRemain : DINT := 1800000;
   Lunch_Min : DINT := 10;
   Lunch_Min_String : STRING_4 := '10';
   Lunch_MinDisplay : DINT := 30;
   Lunch_SecDisplay : DINT;
   Lunch_SecRemain : DINT := 1800;
   Lunch_SecWholeMin : DINT := 1800;
   Lunch_Timer : TIMER := (PRE := 1800000);
   Midnight_Hour : DINT := 24;
   OneShot : DINT;
        .0   // BREAK 1 TRIGGER ONE SHOT
        .1   // BREAK 2 TRIGGER ONE SHOT
        .2   // LUNCH TRIGGER ONE SHOT
        .3   // THEORETICAL UNIT COUNT TRIGGER ONE SHOT
   ONS_20 : DINT;
        .0   // BARCODE READ FROM LODESTAR STATUS ONE SHOT
        .1   // CLEAR BARCODE READ FROM LODESTAR STATUS ONE SHOT
   prevCalculateLocal : DINT := 1;
   PreviousCount : DINT := 681;
   previousSerialNumber : STRING := 'M91940611';
   PreviousShift : DINT;
   readIndex : DINT;
   register : DINT := 5;   // ARRAY POINTER FOR AVERAGE ASSEMBLY TIME ARRAY
   Rotate_MilliRemain : DINT;
   Rotate_Seconds_perShift : DINT;
   Rotate_SecRemain : DINT;
   Shift_Break_Lengths : DINT := 50;
   Shift_Break_Lengths_Remain : DINT := 39;
   Shift_Delay_Min : DINT := 25;
   Shift_Extra_Min : DINT := 5;
   Shift_Hours : DINT := 9;
   Shift_Hours_Remain : DINT := -17;
   Shift_Minutes : DINT := 460;
   Shift_Minutes_Remain : DINT := -1077;
   Shift_Reset : BOOL;
   Shift_Seconds : DINT := 27600;
   Shift_Seconds_Remain : DINT := -64620;
   Start_Hour : DINT := 7;
   Start_Hour_String : STRING_4 := '07';
   Start_Min : DINT := 5;
   Start_Min_String : STRING_4 := '05';
   tempIndex : DINT := 22;
   TestDateTime : DINT;
   theoreticalUnitsReal : REAL;
   writeIndex : DINT;
END_VAR

ROUTINE MainRoutine   (* ladder *)
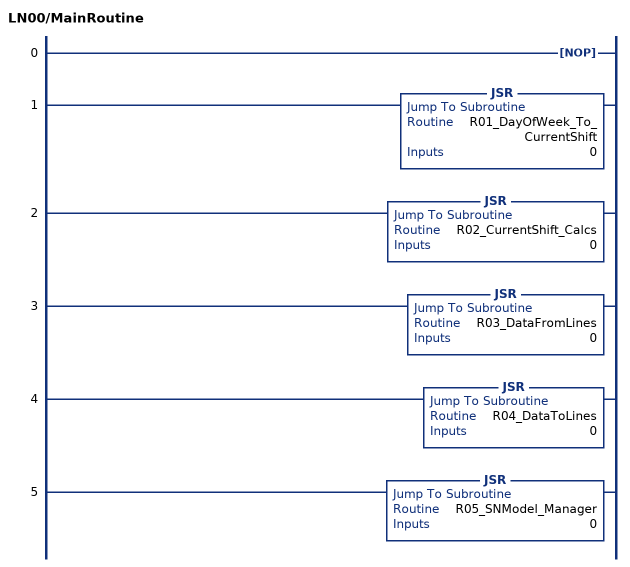
   0: NOP();
   1: JSR(R01_DayOfWeek_To_CurrentShift,0);
   2: JSR(R02_CurrentShift_Calcs,0);
   3: JSR(R03_DataFromLines,0);
   4: JSR(R04_DataToLines,0);
   5: JSR(R05_SNModel_Manager,0);
END_ROUTINE

ROUTINE R01_DayOfWeek_To_CurrentShift   (* ladder *)
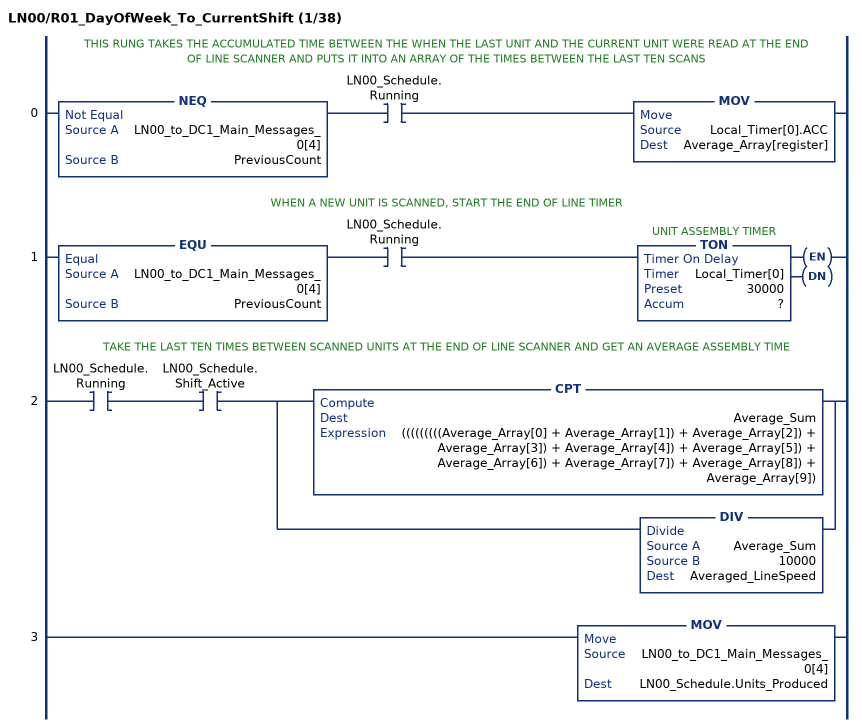
   // THIS RUNG TAKES THE ACCUMULATED TIME BETWEEN THE WHEN THE LAST UNIT AND THE CURRENT UNIT WERE READ AT THE END OF LINE SCANNER AND PUTS IT INTO AN ARRAY OF THE TIMES BETWEEN THE LAST TEN SCANS
   0: NEQ(LN00_to_DC1_Main_Messages_0[4],PreviousCount)XIC(LN00_Schedule.Running)MOV(Local_Timer[0].ACC,Average_Array[register]);
   // WHEN A NEW UNIT IS SCANNED, START THE END OF LINE TIMER
   1: EQU(LN00_to_DC1_Main_Messages_0[4],PreviousCount)XIC(LN00_Schedule.Running)TON(Local_Timer[0],?,?);
   // TAKE THE LAST TEN TIMES BETWEEN SCANNED UNITS AT THE END OF LINE SCANNER AND GET AN AVERAGE ASSEMBLY TIME
   2: XIC(LN00_Schedule.Running)XIC(LN00_Schedule.Shift_Active)[CPT(Average_Sum,(((((((((Average_Array[0] + Average_Array[1]) + Average_Array[2]) + Average_Array[3]) + Average_Array[4]) + Average_Array[5]) + Average_Array[6]) + Average_Array[7]) + Average_Array[8]) + Average_Array[9])) ,DIV(Average_Sum,10000,Averaged_LineSpeed) ];
   3: MOV(LN00_to_DC1_Main_Messages_0[4],LN00_Schedule.Units_Produced);
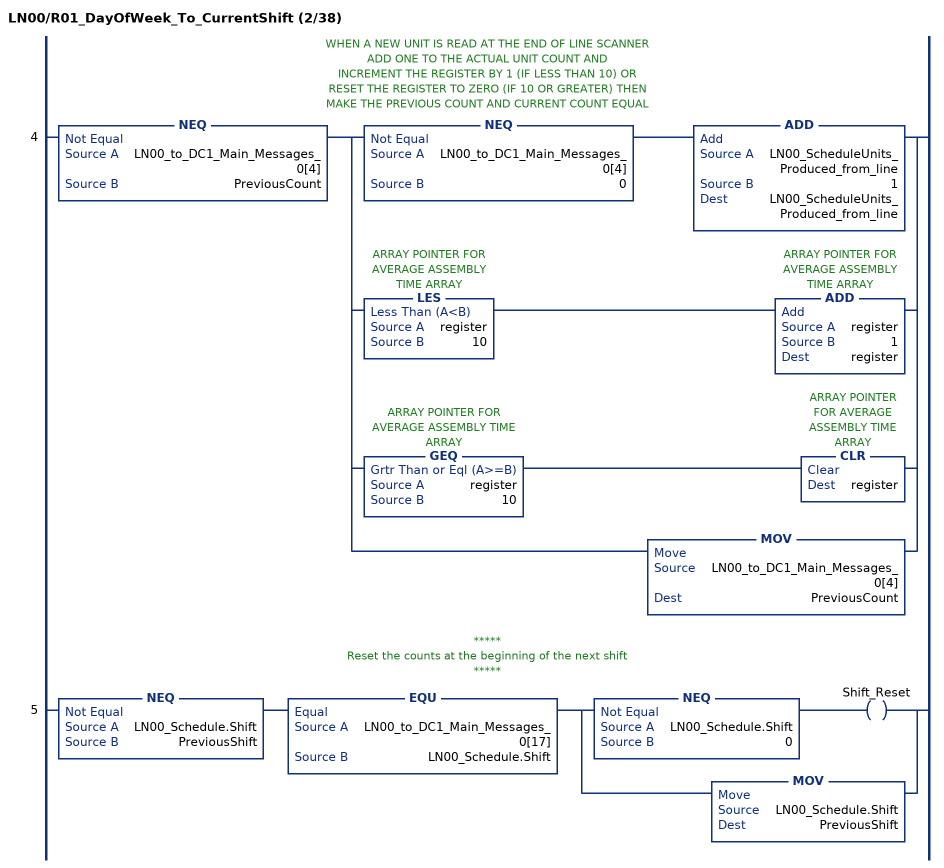
   // WHEN A NEW UNIT IS READ AT THE END OF LINE SCANNER
   // ADD ONE TO THE ACTUAL UNIT COUNT AND
   // INCREMENT THE REGISTER BY 1 (IF LESS THAN 10) OR
   // RESET THE REGISTER TO ZERO (IF 10 OR GREATER) THEN
   // MAKE THE PREVIOUS COUNT AND CURRENT COUNT EQUAL
   4: NEQ(LN00_to_DC1_Main_Messages_0[4],PreviousCount)[NEQ(LN00_to_DC1_Main_Messages_0[4],0) ADD(LN00_ScheduleUnits_Produced_from_line,1,LN00_ScheduleUnits_Produced_from_line) ,LES(register,10) ADD(register,1,register) ,GEQ(register,10) CLR(register) ,MOV(LN00_to_DC1_Main_Messages_0[4],PreviousCount) ];
   // *****
   // Reset the counts at the beginning of the next shift
   // *****
   5: NEQ(LN00_Schedule.Shift,PreviousShift)EQU(LN00_to_DC1_Main_Messages_0[17],LN00_Schedule.Shift)[NEQ(LN00_Schedule.Shift,0) OTE(Shift_Reset) ,MOV(LN00_Schedule.Shift,PreviousShift) ];
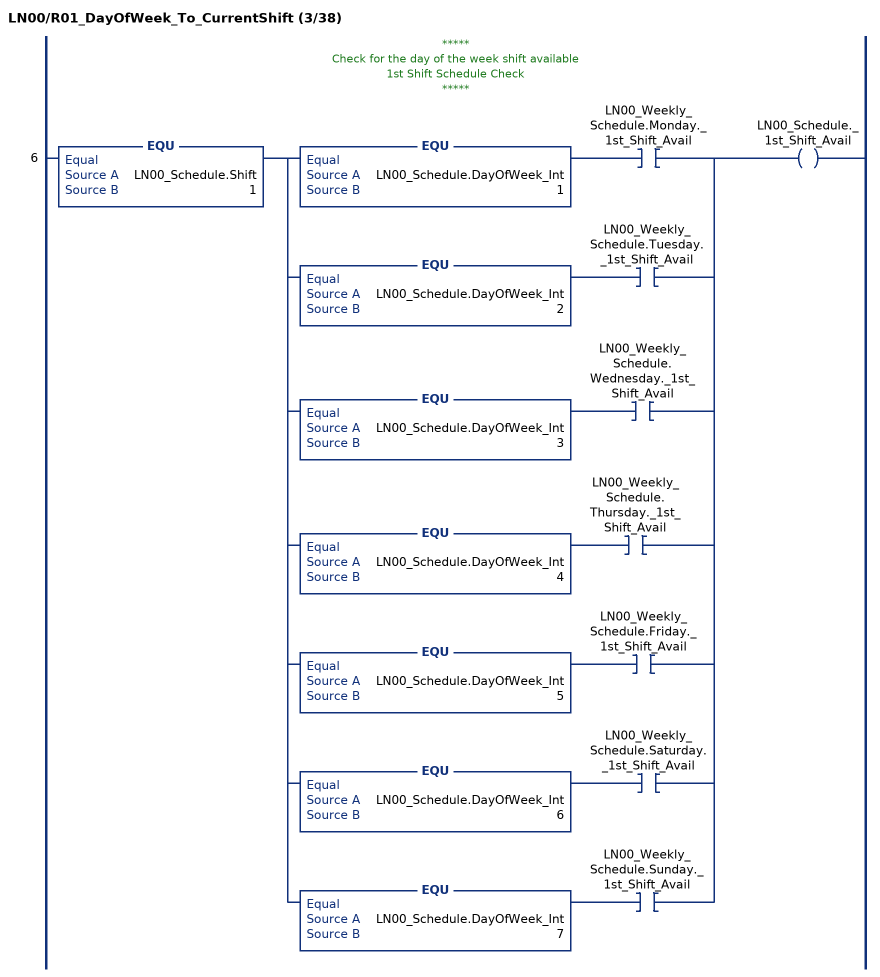
   // *****
   // Check for the day of the week shift available
   // 1st Shift Schedule Check
   // *****
   6: EQU(LN00_Schedule.Shift,1)[EQU(LN00_Schedule.DayOfWeek_Int,1) XIC(LN00_Weekly_Schedule.Monday._1st_Shift_Avail) ,EQU(LN00_Schedule.DayOfWeek_Int,2) XIC(LN00_Weekly_Schedule.Tuesday._1st_Shift_Avail) ,EQU(LN00_Schedule.DayOfWeek_Int,3) XIC(LN00_Weekly_Schedule.Wednesday._1st_Shift_Avail) ,EQU(LN00_Schedule.DayOfWeek_Int,4) XIC(LN00_Weekly_Schedule.Thursday._1st_Shift_Avail) ,EQU(LN00_Schedule.DayOfWeek_Int,5) XIC(LN00_Weekly_Schedule.Friday._1st_Shift_Avail) ,EQU(LN00_Schedule.DayOfWeek_Int,6) XIC(LN00_Weekly_Schedule.Saturday._1st_Shift_Avail) ,EQU(LN00_Schedule.DayOfWeek_Int,7) XIC(LN00_Weekly_Schedule.Sunday._1st_Shift_Avail) ]OTE(LN00_Schedule._1st_Shift_Avail);
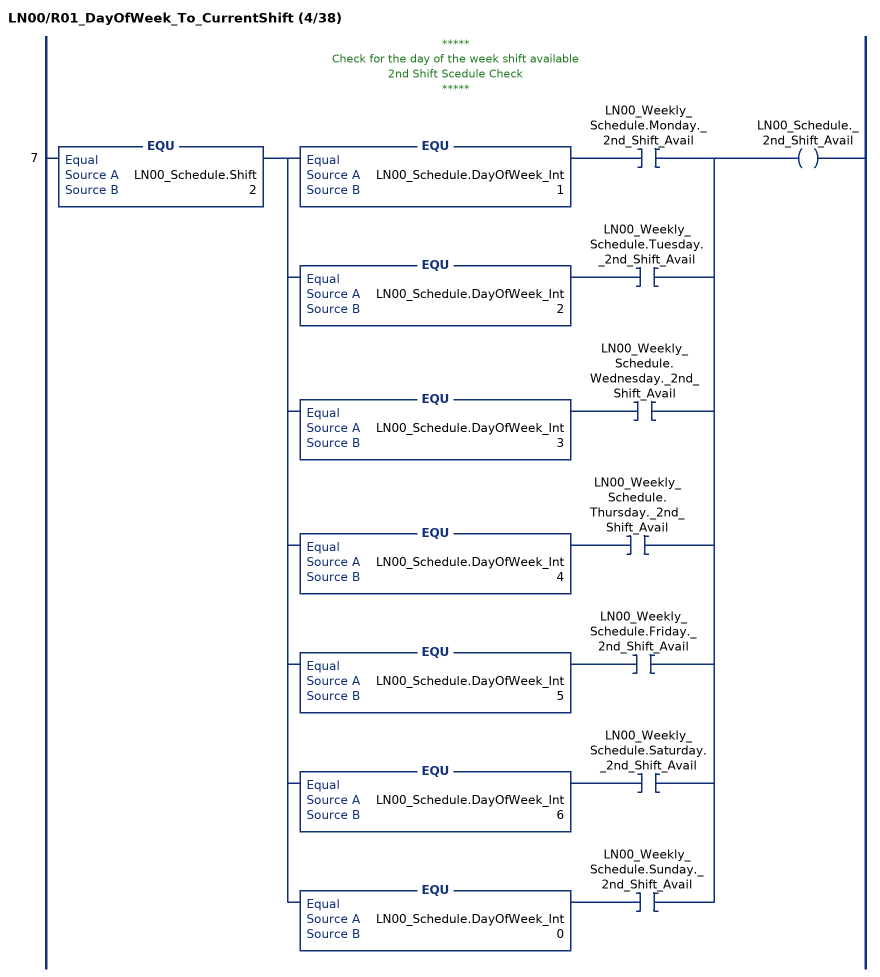
   // *****
   // Check for the day of the week shift available
   // 2nd Shift Scedule Check
   // *****
   7: EQU(LN00_Schedule.Shift,2)[EQU(LN00_Schedule.DayOfWeek_Int,1) XIC(LN00_Weekly_Schedule.Monday._2nd_Shift_Avail) ,EQU(LN00_Schedule.DayOfWeek_Int,2) XIC(LN00_Weekly_Schedule.Tuesday._2nd_Shift_Avail) ,EQU(LN00_Schedule.DayOfWeek_Int,3) XIC(LN00_Weekly_Schedule.Wednesday._2nd_Shift_Avail) ,EQU(LN00_Schedule.DayOfWeek_Int,4) XIC(LN00_Weekly_Schedule.Thursday._2nd_Shift_Avail) ,EQU(LN00_Schedule.DayOfWeek_Int,5) XIC(LN00_Weekly_Schedule.Friday._2nd_Shift_Avail) ,EQU(LN00_Schedule.DayOfWeek_Int,6) XIC(LN00_Weekly_Schedule.Saturday._2nd_Shift_Avail) ,EQU(LN00_Schedule.DayOfWeek_Int,0) XIC(LN00_Weekly_Schedule.Sunday._2nd_Shift_Avail) ]OTE(LN00_Schedule._2nd_Shift_Avail);
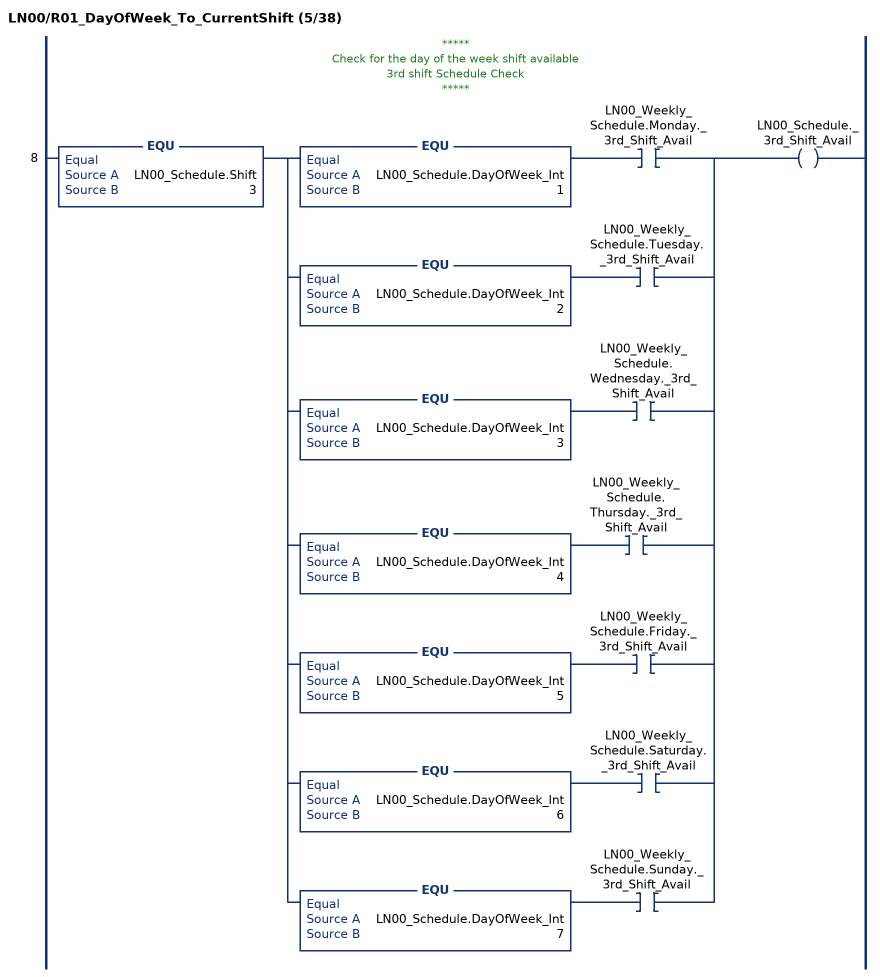
   // *****
   // Check for the day of the week shift available
   // 3rd shift Schedule Check
   // *****
   8: EQU(LN00_Schedule.Shift,3)[EQU(LN00_Schedule.DayOfWeek_Int,1) XIC(LN00_Weekly_Schedule.Monday._3rd_Shift_Avail) ,EQU(LN00_Schedule.DayOfWeek_Int,2) XIC(LN00_Weekly_Schedule.Tuesday._3rd_Shift_Avail) ,EQU(LN00_Schedule.DayOfWeek_Int,3) XIC(LN00_Weekly_Schedule.Wednesday._3rd_Shift_Avail) ,EQU(LN00_Schedule.DayOfWeek_Int,4) XIC(LN00_Weekly_Schedule.Thursday._3rd_Shift_Avail) ,EQU(LN00_Schedule.DayOfWeek_Int,5) XIC(LN00_Weekly_Schedule.Friday._3rd_Shift_Avail) ,EQU(LN00_Schedule.DayOfWeek_Int,6) XIC(LN00_Weekly_Schedule.Saturday._3rd_Shift_Avail) ,EQU(LN00_Schedule.DayOfWeek_Int,7) XIC(LN00_Weekly_Schedule.Sunday._3rd_Shift_Avail) ]OTE(LN00_Schedule._3rd_Shift_Avail);
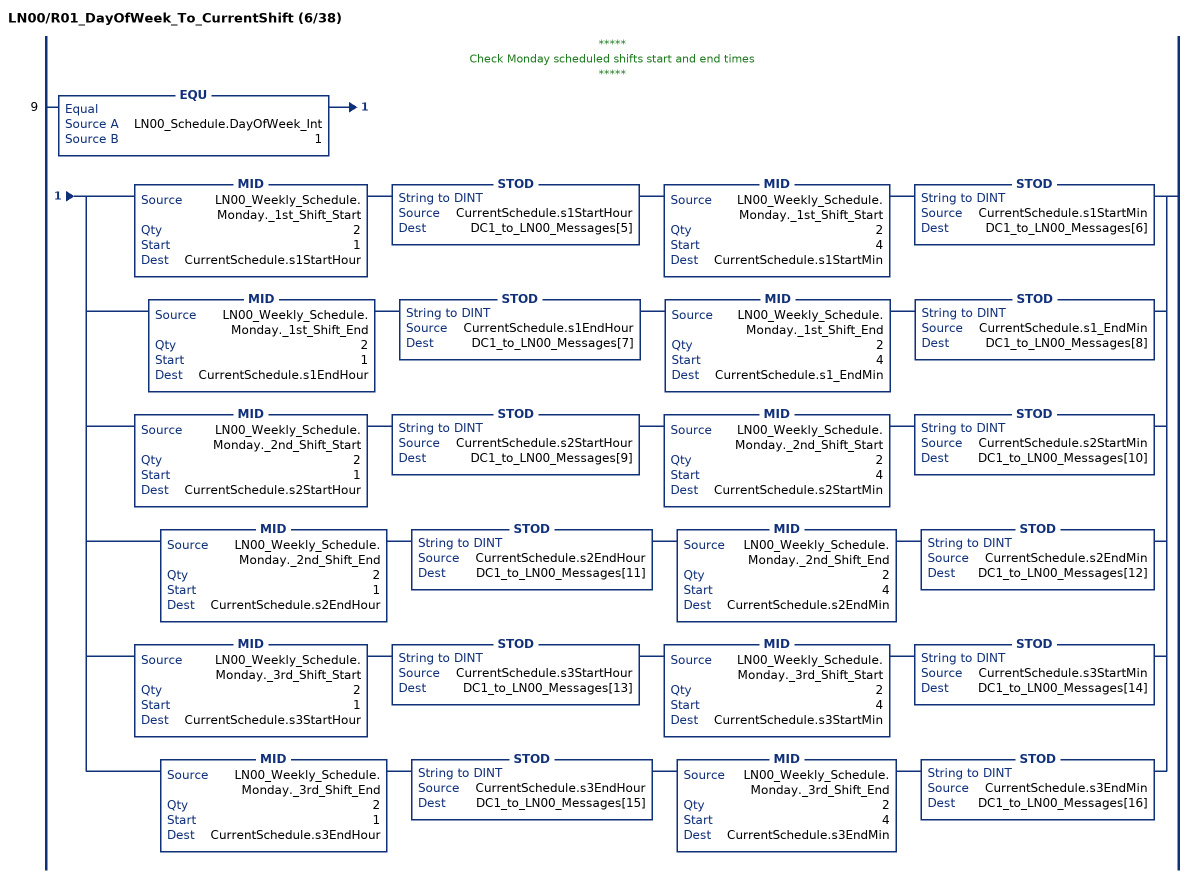
   // *****
   // Check Monday scheduled shifts start and end times
   // *****
   9: EQU(LN00_Schedule.DayOfWeek_Int,1)[MID(LN00_Weekly_Schedule.Monday._1st_Shift_Start,2,1,CurrentSchedule.s1StartHour) STOD(CurrentSchedule.s1StartHour,DC1_to_LN00_Messages[5]) MID(LN00_Weekly_Schedule.Monday._1st_Shift_Start,2,4,CurrentSchedule.s1StartMin) STOD(CurrentSchedule.s1StartMin,DC1_to_LN00_Messages[6]) ,MID(LN00_Weekly_Schedule.Monday._1st_Shift_End,2,1,CurrentSchedule.s1EndHour) STOD(CurrentSchedule.s1EndHour,DC1_to_LN00_Messages[7]) MID(LN00_Weekly_Schedule.Monday._1st_Shift_End,2,4,CurrentSchedule.s1_EndMin) STOD(CurrentSchedule.s1_EndMin,DC1_to_LN00_Messages[8]) ,MID(LN00_Weekly_Schedule.Monday._2nd_Shift_Start,2,1,CurrentSchedule.s2StartHour) STOD(CurrentSchedule.s2StartHour,DC1_to_LN00_Messages[9]) MID(LN00_Weekly_Schedule.Monday._2nd_Shift_Start,2,4,CurrentSchedule.s2StartMin) STOD(CurrentSchedule.s2StartMin,DC1_to_LN00_Messages[10]) ,MID(LN00_Weekly_Schedule.Monday._2nd_Shift_End,2,1,CurrentSchedule.s2EndHour) STOD(CurrentSchedule.s2EndHour,DC1_to_LN00_Messages[11]) MID(LN00_Weekly_Schedule.Monday._2nd_Shift_End,2,4,CurrentSchedule.s2EndMin) STOD(CurrentSchedule.s2EndMin,DC1_to_LN00_Messages[12]) ,MID(LN00_Weekly_Schedule.Monday._3rd_Shift_Start,2,1,CurrentSchedule.s3StartHour) STOD(CurrentSchedule.s3StartHour,DC1_to_LN00_Messages[13]) MID(LN00_Weekly_Schedule.Monday._3rd_Shift_Start,2,4,CurrentSchedule.s3StartMin) STOD(CurrentSchedule.s3StartMin,DC1_to_LN00_Messages[14]) ,MID(LN00_Weekly_Schedule.Monday._3rd_Shift_End,2,1,CurrentSchedule.s3EndHour) STOD(CurrentSchedule.s3EndHour,DC1_to_LN00_Messages[15]) MID(LN00_Weekly_Schedule.Monday._3rd_Shift_End,2,4,CurrentSchedule.s3EndMin) STOD(CurrentSchedule.s3EndMin,DC1_to_LN00_Messages[16]) ];
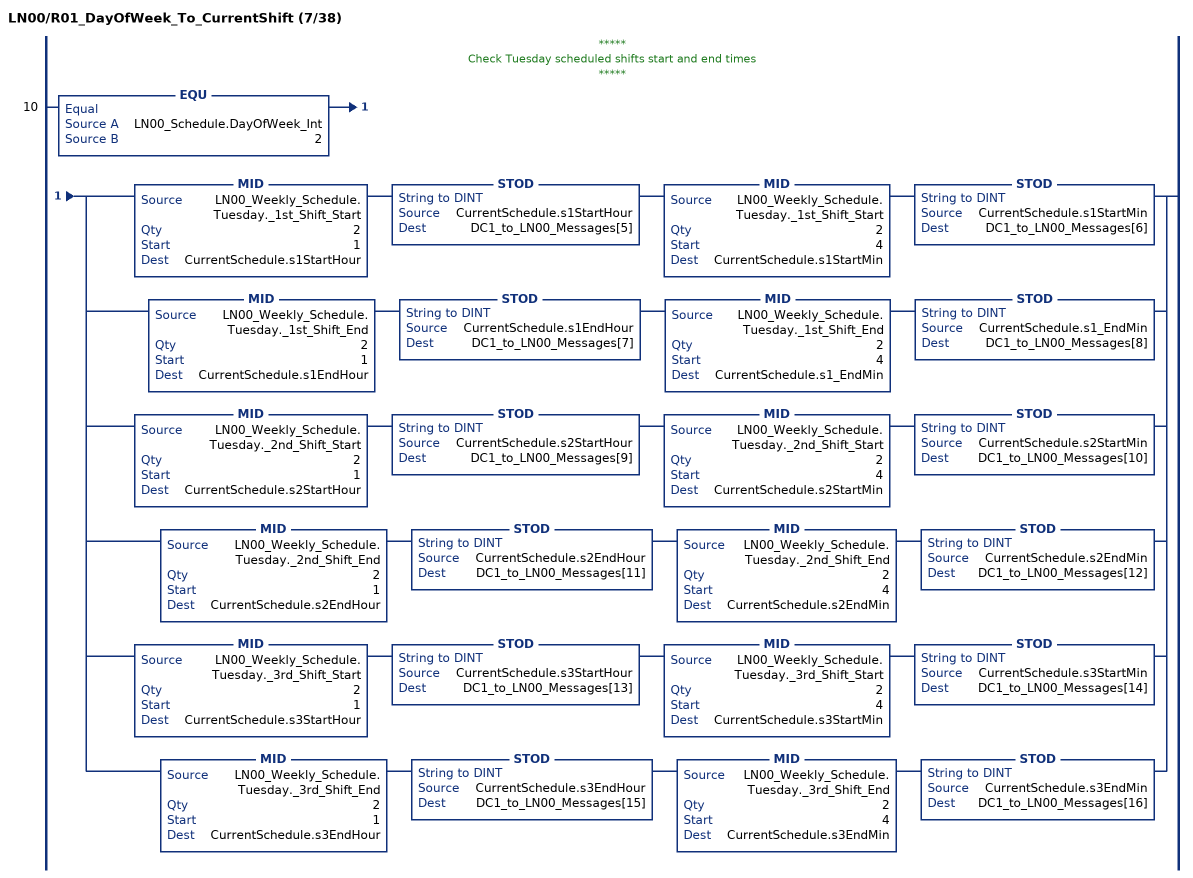
   // *****
   // Check Tuesday scheduled shifts start and end times
   // *****
   10: EQU(LN00_Schedule.DayOfWeek_Int,2)[MID(LN00_Weekly_Schedule.Tuesday._1st_Shift_Start,2,1,CurrentSchedule.s1StartHour) STOD(CurrentSchedule.s1StartHour,DC1_to_LN00_Messages[5]) MID(LN00_Weekly_Schedule.Tuesday._1st_Shift_Start,2,4,CurrentSchedule.s1StartMin) STOD(CurrentSchedule.s1StartMin,DC1_to_LN00_Messages[6]) ,MID(LN00_Weekly_Schedule.Tuesday._1st_Shift_End,2,1,CurrentSchedule.s1EndHour) STOD(CurrentSchedule.s1EndHour,DC1_to_LN00_Messages[7]) MID(LN00_Weekly_Schedule.Tuesday._1st_Shift_End,2,4,CurrentSchedule.s1_EndMin) STOD(CurrentSchedule.s1_EndMin,DC1_to_LN00_Messages[8]) ,MID(LN00_Weekly_Schedule.Tuesday._2nd_Shift_Start,2,1,CurrentSchedule.s2StartHour) STOD(CurrentSchedule.s2StartHour,DC1_to_LN00_Messages[9]) MID(LN00_Weekly_Schedule.Tuesday._2nd_Shift_Start,2,4,CurrentSchedule.s2StartMin) STOD(CurrentSchedule.s2StartMin,DC1_to_LN00_Messages[10]) ,MID(LN00_Weekly_Schedule.Tuesday._2nd_Shift_End,2,1,CurrentSchedule.s2EndHour) STOD(CurrentSchedule.s2EndHour,DC1_to_LN00_Messages[11]) MID(LN00_Weekly_Schedule.Tuesday._2nd_Shift_End,2,4,CurrentSchedule.s2EndMin) STOD(CurrentSchedule.s2EndMin,DC1_to_LN00_Messages[12]) ,MID(LN00_Weekly_Schedule.Tuesday._3rd_Shift_Start,2,1,CurrentSchedule.s3StartHour) STOD(CurrentSchedule.s3StartHour,DC1_to_LN00_Messages[13]) MID(LN00_Weekly_Schedule.Tuesday._3rd_Shift_Start,2,4,CurrentSchedule.s3StartMin) STOD(CurrentSchedule.s3StartMin,DC1_to_LN00_Messages[14]) ,MID(LN00_Weekly_Schedule.Tuesday._3rd_Shift_End,2,1,CurrentSchedule.s3EndHour) STOD(CurrentSchedule.s3EndHour,DC1_to_LN00_Messages[15]) MID(LN00_Weekly_Schedule.Tuesday._3rd_Shift_End,2,4,CurrentSchedule.s3EndMin) STOD(CurrentSchedule.s3EndMin,DC1_to_LN00_Messages[16]) ];
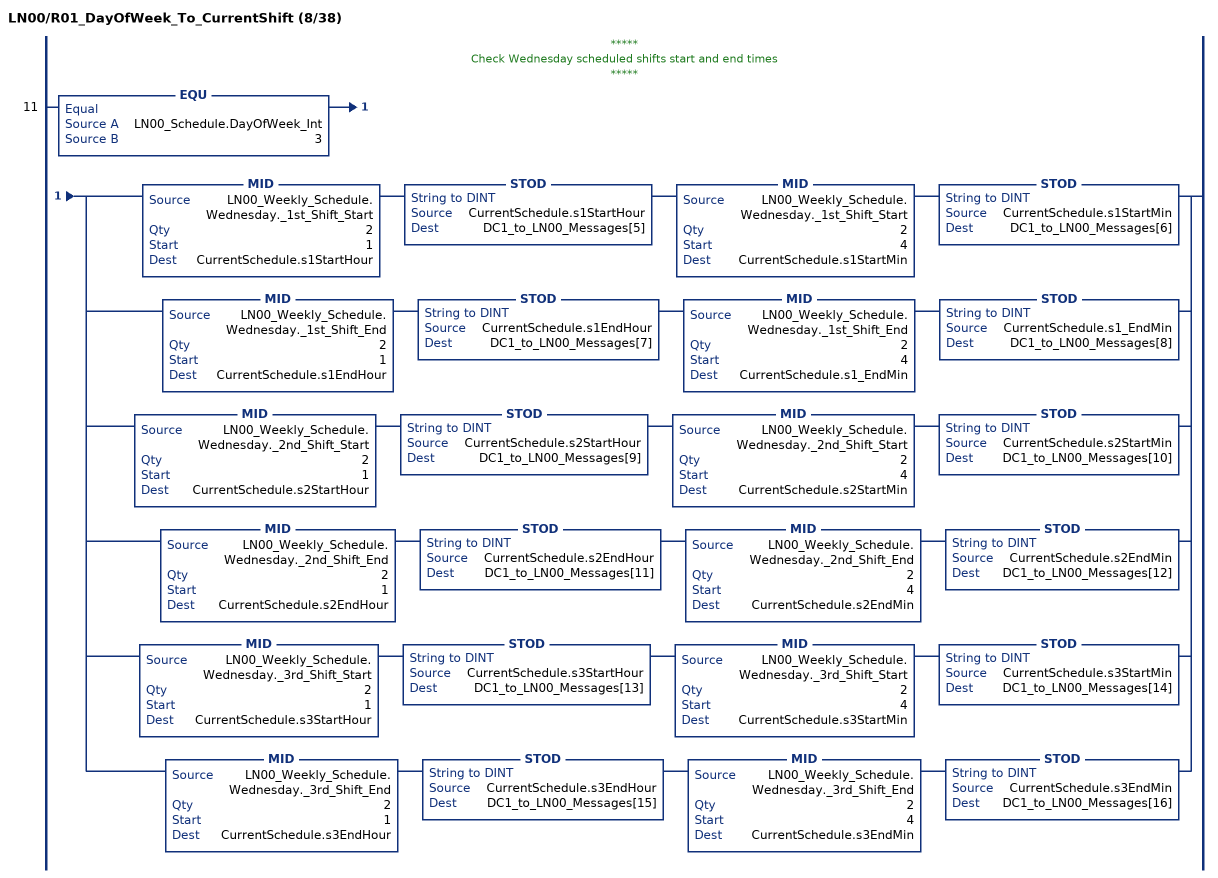
   // *****
   // Check Wednesday scheduled shifts start and end times
   // *****
   11: EQU(LN00_Schedule.DayOfWeek_Int,3)[MID(LN00_Weekly_Schedule.Wednesday._1st_Shift_Start,2,1,CurrentSchedule.s1StartHour) STOD(CurrentSchedule.s1StartHour,DC1_to_LN00_Messages[5]) MID(LN00_Weekly_Schedule.Wednesday._1st_Shift_Start,2,4,CurrentSchedule.s1StartMin) STOD(CurrentSchedule.s1StartMin,DC1_to_LN00_Messages[6]) ,MID(LN00_Weekly_Schedule.Wednesday._1st_Shift_End,2,1,CurrentSchedule.s1EndHour) STOD(CurrentSchedule.s1EndHour,DC1_to_LN00_Messages[7]) MID(LN00_Weekly_Schedule.Wednesday._1st_Shift_End,2,4,CurrentSchedule.s1_EndMin) STOD(CurrentSchedule.s1_EndMin,DC1_to_LN00_Messages[8]) ,MID(LN00_Weekly_Schedule.Wednesday._2nd_Shift_Start,2,1,CurrentSchedule.s2StartHour) STOD(CurrentSchedule.s2StartHour,DC1_to_LN00_Messages[9]) MID(LN00_Weekly_Schedule.Wednesday._2nd_Shift_Start,2,4,CurrentSchedule.s2StartMin) STOD(CurrentSchedule.s2StartMin,DC1_to_LN00_Messages[10]) ,MID(LN00_Weekly_Schedule.Wednesday._2nd_Shift_End,2,1,CurrentSchedule.s2EndHour) STOD(CurrentSchedule.s2EndHour,DC1_to_LN00_Messages[11]) MID(LN00_Weekly_Schedule.Wednesday._2nd_Shift_End,2,4,CurrentSchedule.s2EndMin) STOD(CurrentSchedule.s2EndMin,DC1_to_LN00_Messages[12]) ,MID(LN00_Weekly_Schedule.Wednesday._3rd_Shift_Start,2,1,CurrentSchedule.s3StartHour) STOD(CurrentSchedule.s3StartHour,DC1_to_LN00_Messages[13]) MID(LN00_Weekly_Schedule.Wednesday._3rd_Shift_Start,2,4,CurrentSchedule.s3StartMin) STOD(CurrentSchedule.s3StartMin,DC1_to_LN00_Messages[14]) ,MID(LN00_Weekly_Schedule.Wednesday._3rd_Shift_End,2,1,CurrentSchedule.s3EndHour) STOD(CurrentSchedule.s3EndHour,DC1_to_LN00_Messages[15]) MID(LN00_Weekly_Schedule.Wednesday._3rd_Shift_End,2,4,CurrentSchedule.s3EndMin) STOD(CurrentSchedule.s3EndMin,DC1_to_LN00_Messages[16]) ];
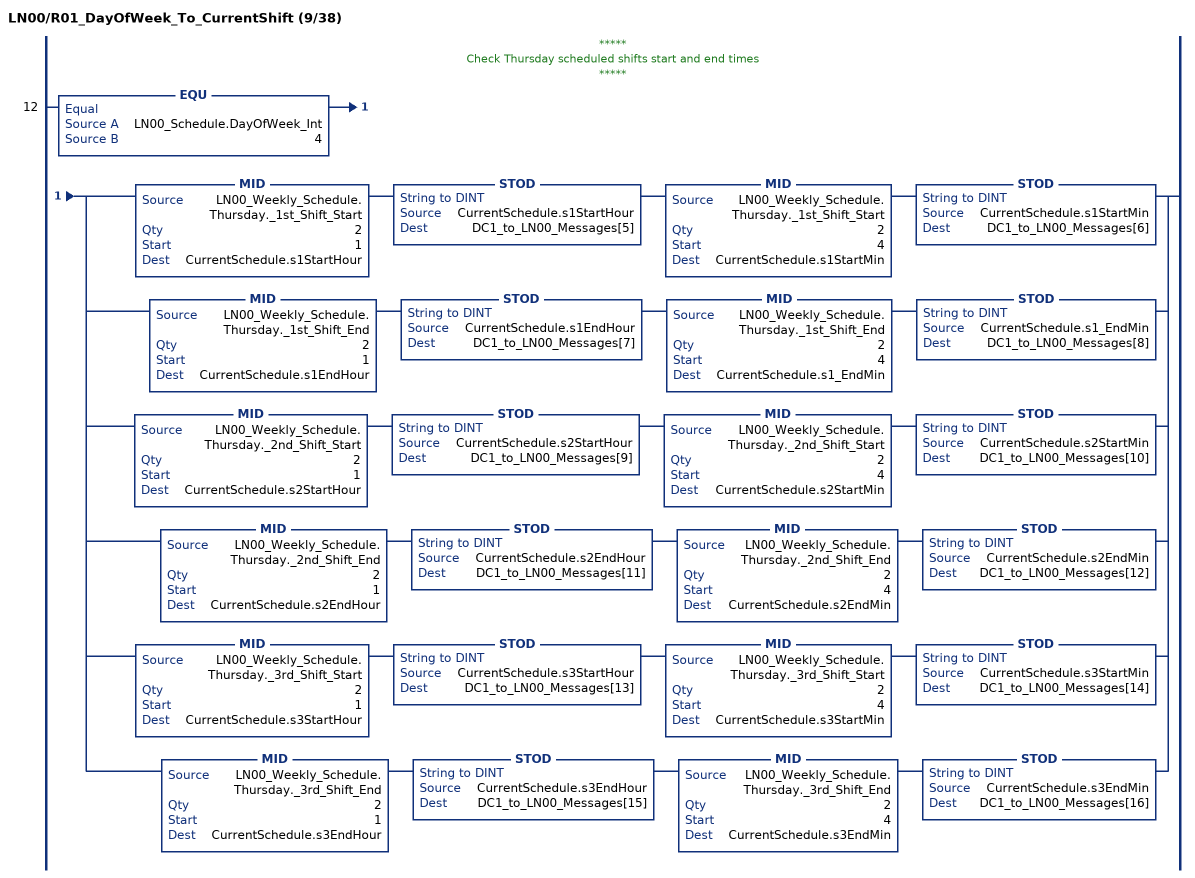
   // *****
   // Check Thursday scheduled shifts start and end times
   // *****
   12: EQU(LN00_Schedule.DayOfWeek_Int,4)[MID(LN00_Weekly_Schedule.Thursday._1st_Shift_Start,2,1,CurrentSchedule.s1StartHour) STOD(CurrentSchedule.s1StartHour,DC1_to_LN00_Messages[5]) MID(LN00_Weekly_Schedule.Thursday._1st_Shift_Start,2,4,CurrentSchedule.s1StartMin) STOD(CurrentSchedule.s1StartMin,DC1_to_LN00_Messages[6]) ,MID(LN00_Weekly_Schedule.Thursday._1st_Shift_End,2,1,CurrentSchedule.s1EndHour) STOD(CurrentSchedule.s1EndHour,DC1_to_LN00_Messages[7]) MID(LN00_Weekly_Schedule.Thursday._1st_Shift_End,2,4,CurrentSchedule.s1_EndMin) STOD(CurrentSchedule.s1_EndMin,DC1_to_LN00_Messages[8]) ,MID(LN00_Weekly_Schedule.Thursday._2nd_Shift_Start,2,1,CurrentSchedule.s2StartHour) STOD(CurrentSchedule.s2StartHour,DC1_to_LN00_Messages[9]) MID(LN00_Weekly_Schedule.Thursday._2nd_Shift_Start,2,4,CurrentSchedule.s2StartMin) STOD(CurrentSchedule.s2StartMin,DC1_to_LN00_Messages[10]) ,MID(LN00_Weekly_Schedule.Thursday._2nd_Shift_End,2,1,CurrentSchedule.s2EndHour) STOD(CurrentSchedule.s2EndHour,DC1_to_LN00_Messages[11]) MID(LN00_Weekly_Schedule.Thursday._2nd_Shift_End,2,4,CurrentSchedule.s2EndMin) STOD(CurrentSchedule.s2EndMin,DC1_to_LN00_Messages[12]) ,MID(LN00_Weekly_Schedule.Thursday._3rd_Shift_Start,2,1,CurrentSchedule.s3StartHour) STOD(CurrentSchedule.s3StartHour,DC1_to_LN00_Messages[13]) MID(LN00_Weekly_Schedule.Thursday._3rd_Shift_Start,2,4,CurrentSchedule.s3StartMin) STOD(CurrentSchedule.s3StartMin,DC1_to_LN00_Messages[14]) ,MID(LN00_Weekly_Schedule.Thursday._3rd_Shift_End,2,1,CurrentSchedule.s3EndHour) STOD(CurrentSchedule.s3EndHour,DC1_to_LN00_Messages[15]) MID(LN00_Weekly_Schedule.Thursday._3rd_Shift_End,2,4,CurrentSchedule.s3EndMin) STOD(CurrentSchedule.s3EndMin,DC1_to_LN00_Messages[16]) ];
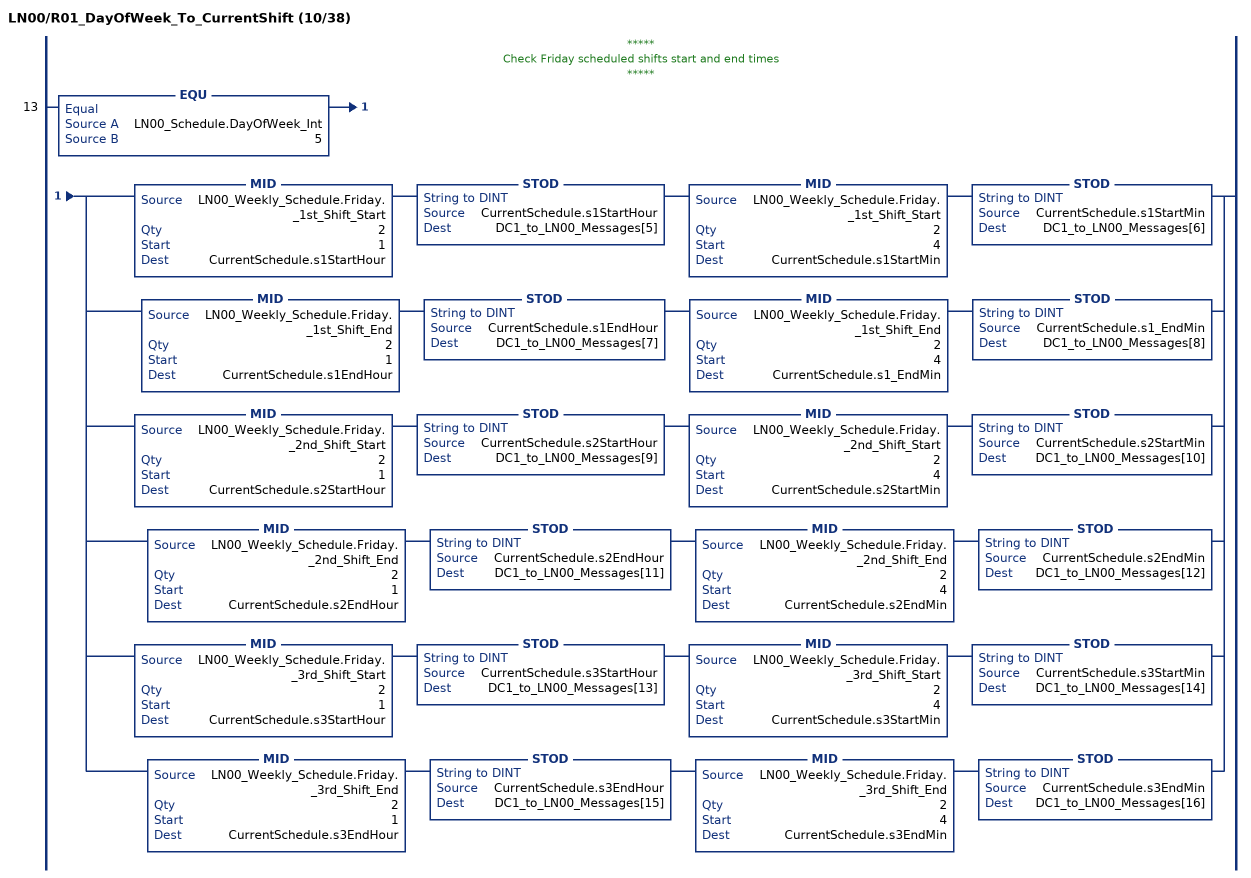
   // *****
   // Check Friday scheduled shifts start and end times
   // *****
   13: EQU(LN00_Schedule.DayOfWeek_Int,5)[MID(LN00_Weekly_Schedule.Friday._1st_Shift_Start,2,1,CurrentSchedule.s1StartHour) STOD(CurrentSchedule.s1StartHour,DC1_to_LN00_Messages[5]) MID(LN00_Weekly_Schedule.Friday._1st_Shift_Start,2,4,CurrentSchedule.s1StartMin) STOD(CurrentSchedule.s1StartMin,DC1_to_LN00_Messages[6]) ,MID(LN00_Weekly_Schedule.Friday._1st_Shift_End,2,1,CurrentSchedule.s1EndHour) STOD(CurrentSchedule.s1EndHour,DC1_to_LN00_Messages[7]) MID(LN00_Weekly_Schedule.Friday._1st_Shift_End,2,4,CurrentSchedule.s1_EndMin) STOD(CurrentSchedule.s1_EndMin,DC1_to_LN00_Messages[8]) ,MID(LN00_Weekly_Schedule.Friday._2nd_Shift_Start,2,1,CurrentSchedule.s2StartHour) STOD(CurrentSchedule.s2StartHour,DC1_to_LN00_Messages[9]) MID(LN00_Weekly_Schedule.Friday._2nd_Shift_Start,2,4,CurrentSchedule.s2StartMin) STOD(CurrentSchedule.s2StartMin,DC1_to_LN00_Messages[10]) ,MID(LN00_Weekly_Schedule.Friday._2nd_Shift_End,2,1,CurrentSchedule.s2EndHour) STOD(CurrentSchedule.s2EndHour,DC1_to_LN00_Messages[11]) MID(LN00_Weekly_Schedule.Friday._2nd_Shift_End,2,4,CurrentSchedule.s2EndMin) STOD(CurrentSchedule.s2EndMin,DC1_to_LN00_Messages[12]) ,MID(LN00_Weekly_Schedule.Friday._3rd_Shift_Start,2,1,CurrentSchedule.s3StartHour) STOD(CurrentSchedule.s3StartHour,DC1_to_LN00_Messages[13]) MID(LN00_Weekly_Schedule.Friday._3rd_Shift_Start,2,4,CurrentSchedule.s3StartMin) STOD(CurrentSchedule.s3StartMin,DC1_to_LN00_Messages[14]) ,MID(LN00_Weekly_Schedule.Friday._3rd_Shift_End,2,1,CurrentSchedule.s3EndHour) STOD(CurrentSchedule.s3EndHour,DC1_to_LN00_Messages[15]) MID(LN00_Weekly_Schedule.Friday._3rd_Shift_End,2,4,CurrentSchedule.s3EndMin) STOD(CurrentSchedule.s3EndMin,DC1_to_LN00_Messages[16]) ];
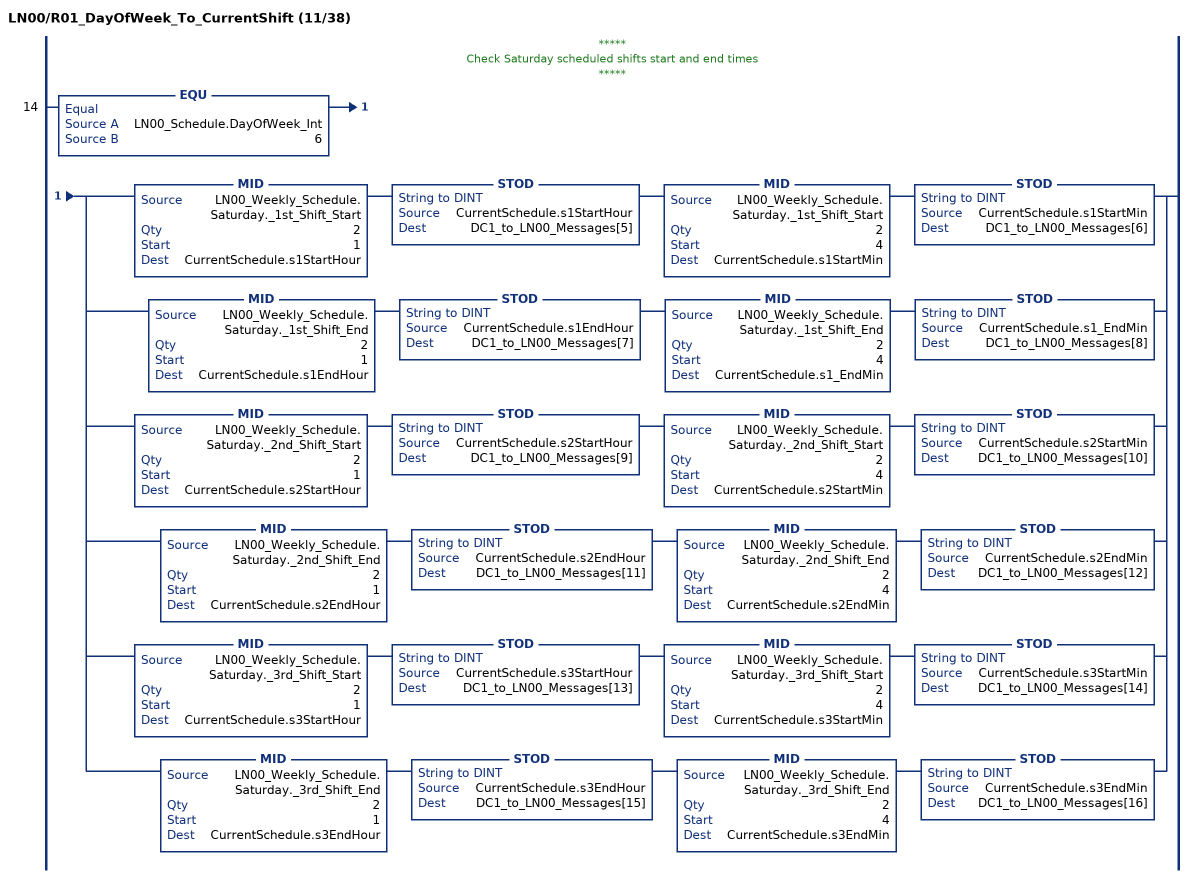
   // *****
   // Check Saturday scheduled shifts start and end times
   // *****
   14: EQU(LN00_Schedule.DayOfWeek_Int,6)[MID(LN00_Weekly_Schedule.Saturday._1st_Shift_Start,2,1,CurrentSchedule.s1StartHour) STOD(CurrentSchedule.s1StartHour,DC1_to_LN00_Messages[5]) MID(LN00_Weekly_Schedule.Saturday._1st_Shift_Start,2,4,CurrentSchedule.s1StartMin) STOD(CurrentSchedule.s1StartMin,DC1_to_LN00_Messages[6]) ,MID(LN00_Weekly_Schedule.Saturday._1st_Shift_End,2,1,CurrentSchedule.s1EndHour) STOD(CurrentSchedule.s1EndHour,DC1_to_LN00_Messages[7]) MID(LN00_Weekly_Schedule.Saturday._1st_Shift_End,2,4,CurrentSchedule.s1_EndMin) STOD(CurrentSchedule.s1_EndMin,DC1_to_LN00_Messages[8]) ,MID(LN00_Weekly_Schedule.Saturday._2nd_Shift_Start,2,1,CurrentSchedule.s2StartHour) STOD(CurrentSchedule.s2StartHour,DC1_to_LN00_Messages[9]) MID(LN00_Weekly_Schedule.Saturday._2nd_Shift_Start,2,4,CurrentSchedule.s2StartMin) STOD(CurrentSchedule.s2StartMin,DC1_to_LN00_Messages[10]) ,MID(LN00_Weekly_Schedule.Saturday._2nd_Shift_End,2,1,CurrentSchedule.s2EndHour) STOD(CurrentSchedule.s2EndHour,DC1_to_LN00_Messages[11]) MID(LN00_Weekly_Schedule.Saturday._2nd_Shift_End,2,4,CurrentSchedule.s2EndMin) STOD(CurrentSchedule.s2EndMin,DC1_to_LN00_Messages[12]) ,MID(LN00_Weekly_Schedule.Saturday._3rd_Shift_Start,2,1,CurrentSchedule.s3StartHour) STOD(CurrentSchedule.s3StartHour,DC1_to_LN00_Messages[13]) MID(LN00_Weekly_Schedule.Saturday._3rd_Shift_Start,2,4,CurrentSchedule.s3StartMin) STOD(CurrentSchedule.s3StartMin,DC1_to_LN00_Messages[14]) ,MID(LN00_Weekly_Schedule.Saturday._3rd_Shift_End,2,1,CurrentSchedule.s3EndHour) STOD(CurrentSchedule.s3EndHour,DC1_to_LN00_Messages[15]) MID(LN00_Weekly_Schedule.Saturday._3rd_Shift_End,2,4,CurrentSchedule.s3EndMin) STOD(CurrentSchedule.s3EndMin,DC1_to_LN00_Messages[16]) ];
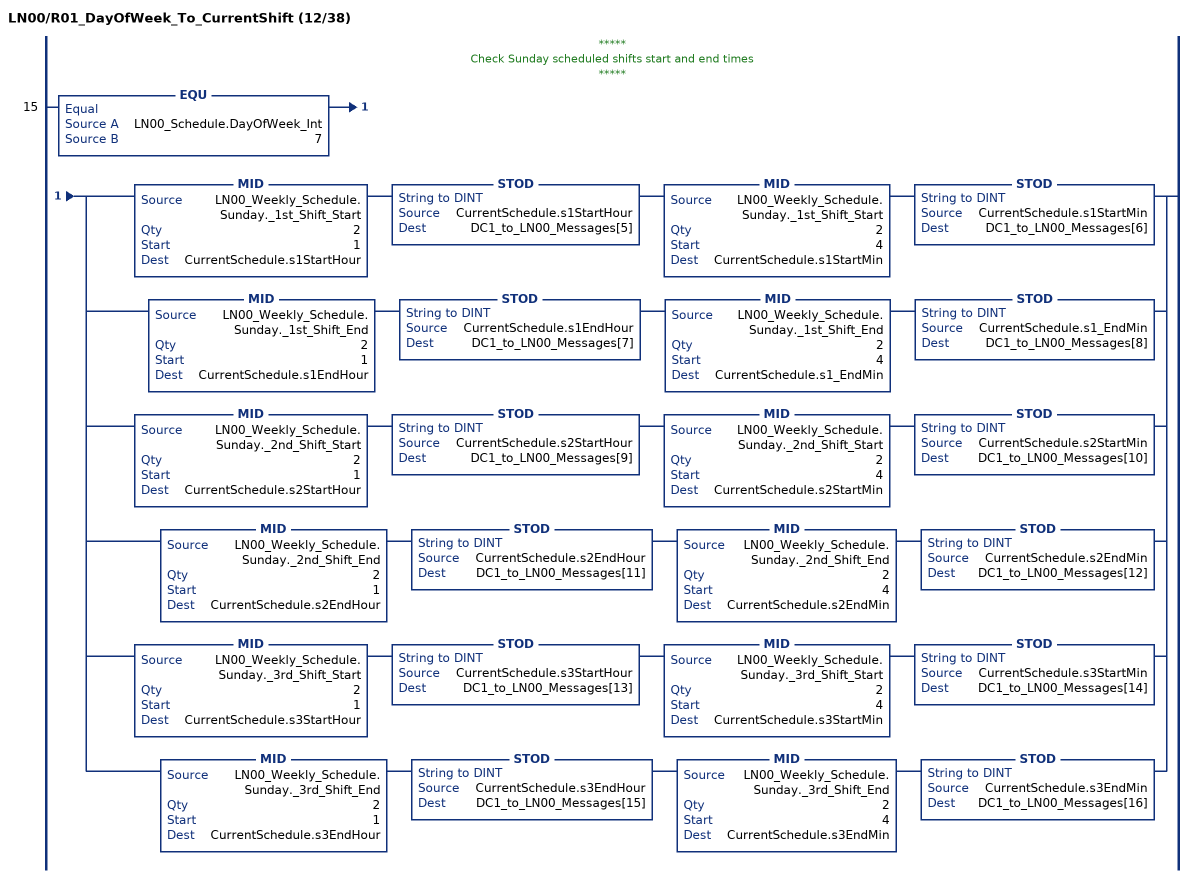
   // *****
   // Check Sunday scheduled shifts start and end times
   // *****
   15: EQU(LN00_Schedule.DayOfWeek_Int,7)[MID(LN00_Weekly_Schedule.Sunday._1st_Shift_Start,2,1,CurrentSchedule.s1StartHour) STOD(CurrentSchedule.s1StartHour,DC1_to_LN00_Messages[5]) MID(LN00_Weekly_Schedule.Sunday._1st_Shift_Start,2,4,CurrentSchedule.s1StartMin) STOD(CurrentSchedule.s1StartMin,DC1_to_LN00_Messages[6]) ,MID(LN00_Weekly_Schedule.Sunday._1st_Shift_End,2,1,CurrentSchedule.s1EndHour) STOD(CurrentSchedule.s1EndHour,DC1_to_LN00_Messages[7]) MID(LN00_Weekly_Schedule.Sunday._1st_Shift_End,2,4,CurrentSchedule.s1_EndMin) STOD(CurrentSchedule.s1_EndMin,DC1_to_LN00_Messages[8]) ,MID(LN00_Weekly_Schedule.Sunday._2nd_Shift_Start,2,1,CurrentSchedule.s2StartHour) STOD(CurrentSchedule.s2StartHour,DC1_to_LN00_Messages[9]) MID(LN00_Weekly_Schedule.Sunday._2nd_Shift_Start,2,4,CurrentSchedule.s2StartMin) STOD(CurrentSchedule.s2StartMin,DC1_to_LN00_Messages[10]) ,MID(LN00_Weekly_Schedule.Sunday._2nd_Shift_End,2,1,CurrentSchedule.s2EndHour) STOD(CurrentSchedule.s2EndHour,DC1_to_LN00_Messages[11]) MID(LN00_Weekly_Schedule.Sunday._2nd_Shift_End,2,4,CurrentSchedule.s2EndMin) STOD(CurrentSchedule.s2EndMin,DC1_to_LN00_Messages[12]) ,MID(LN00_Weekly_Schedule.Sunday._3rd_Shift_Start,2,1,CurrentSchedule.s3StartHour) STOD(CurrentSchedule.s3StartHour,DC1_to_LN00_Messages[13]) MID(LN00_Weekly_Schedule.Sunday._3rd_Shift_Start,2,4,CurrentSchedule.s3StartMin) STOD(CurrentSchedule.s3StartMin,DC1_to_LN00_Messages[14]) ,MID(LN00_Weekly_Schedule.Sunday._3rd_Shift_End,2,1,CurrentSchedule.s3EndHour) STOD(CurrentSchedule.s3EndHour,DC1_to_LN00_Messages[15]) MID(LN00_Weekly_Schedule.Sunday._3rd_Shift_End,2,4,CurrentSchedule.s3EndMin) STOD(CurrentSchedule.s3EndMin,DC1_to_LN00_Messages[16]) ];
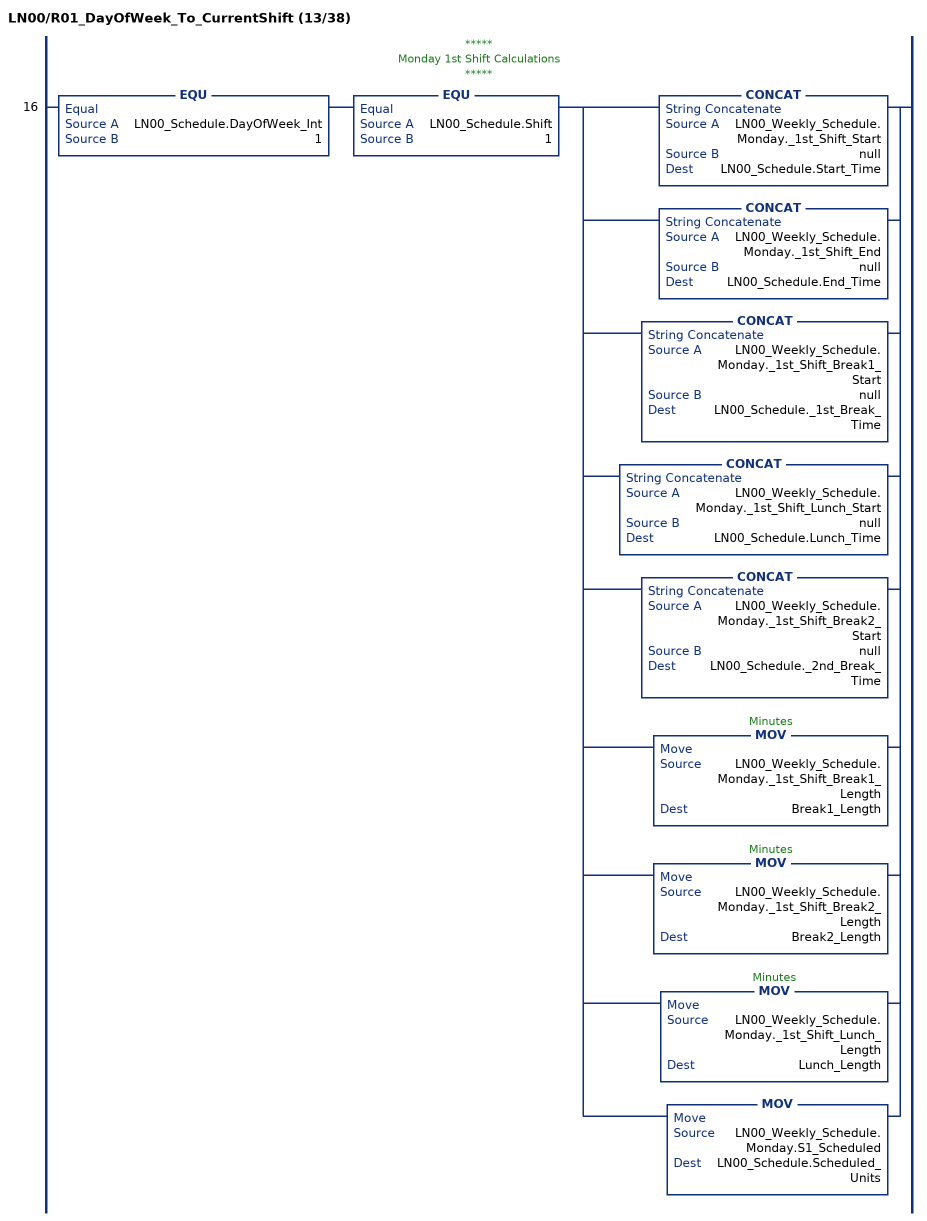
   // *****
   // Monday 1st Shift Calculations
   // *****
   16: EQU(LN00_Schedule.DayOfWeek_Int,1)EQU(LN00_Schedule.Shift,1)[CONCAT(LN00_Weekly_Schedule.Monday._1st_Shift_Start,null,LN00_Schedule.Start_Time) ,CONCAT(LN00_Weekly_Schedule.Monday._1st_Shift_End,null,LN00_Schedule.End_Time) ,CONCAT(LN00_Weekly_Schedule.Monday._1st_Shift_Break1_Start,null,LN00_Schedule._1st_Break_Time) ,CONCAT(LN00_Weekly_Schedule.Monday._1st_Shift_Lunch_Start,null,LN00_Schedule.Lunch_Time) ,CONCAT(LN00_Weekly_Schedule.Monday._1st_Shift_Break2_Start,null,LN00_Schedule._2nd_Break_Time) ,MOV(LN00_Weekly_Schedule.Monday._1st_Shift_Break1_Length,Break1_Length) ,MOV(LN00_Weekly_Schedule.Monday._1st_Shift_Break2_Length,Break2_Length) ,MOV(LN00_Weekly_Schedule.Monday._1st_Shift_Lunch_Length,Lunch_Length) ,MOV(LN00_Weekly_Schedule.Monday.S1_Scheduled,LN00_Schedule.Scheduled_Units) ];
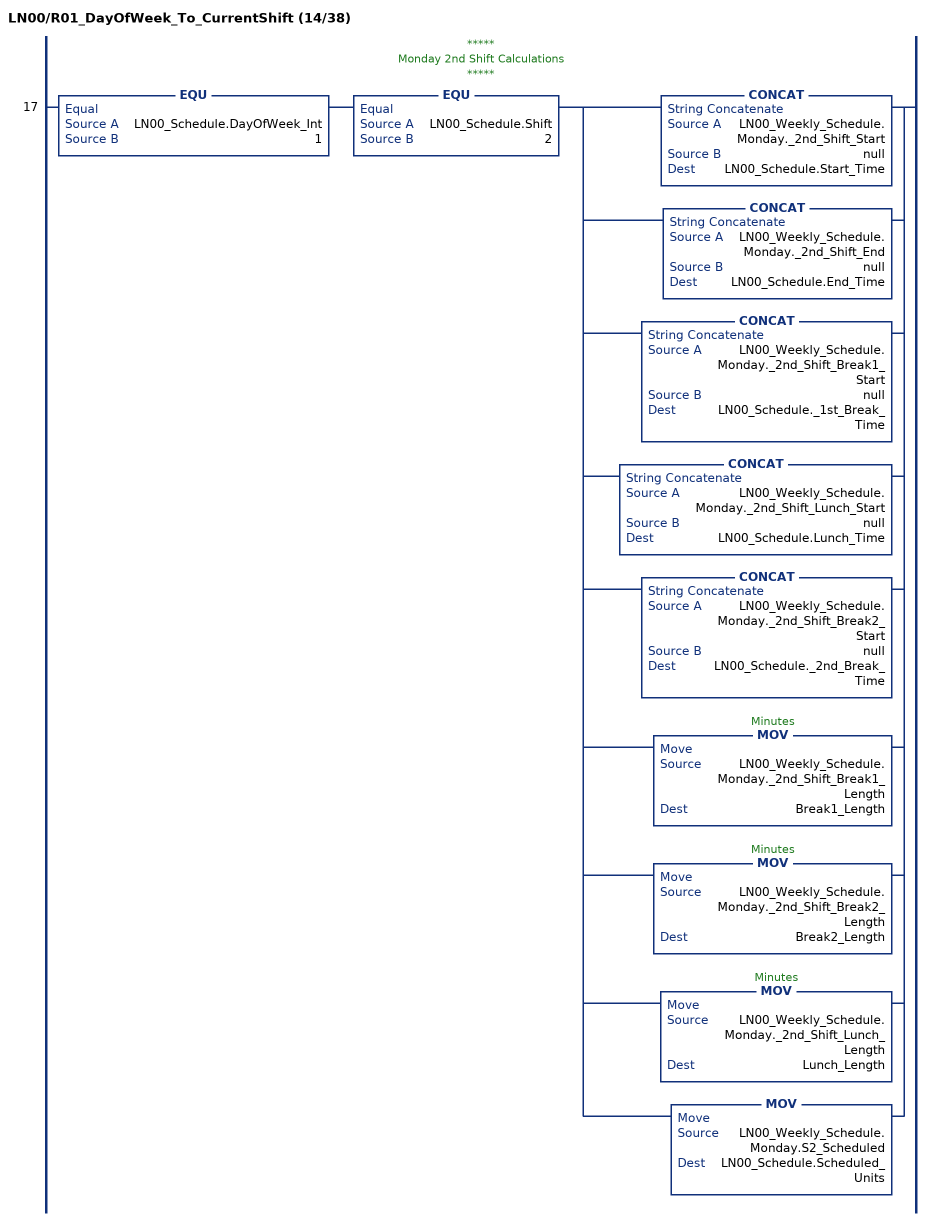
   // *****
   // Monday 2nd Shift Calculations
   // *****
   17: EQU(LN00_Schedule.DayOfWeek_Int,1)EQU(LN00_Schedule.Shift,2)[CONCAT(LN00_Weekly_Schedule.Monday._2nd_Shift_Start,null,LN00_Schedule.Start_Time) ,CONCAT(LN00_Weekly_Schedule.Monday._2nd_Shift_End,null,LN00_Schedule.End_Time) ,CONCAT(LN00_Weekly_Schedule.Monday._2nd_Shift_Break1_Start,null,LN00_Schedule._1st_Break_Time) ,CONCAT(LN00_Weekly_Schedule.Monday._2nd_Shift_Lunch_Start,null,LN00_Schedule.Lunch_Time) ,CONCAT(LN00_Weekly_Schedule.Monday._2nd_Shift_Break2_Start,null,LN00_Schedule._2nd_Break_Time) ,MOV(LN00_Weekly_Schedule.Monday._2nd_Shift_Break1_Length,Break1_Length) ,MOV(LN00_Weekly_Schedule.Monday._2nd_Shift_Break2_Length,Break2_Length) ,MOV(LN00_Weekly_Schedule.Monday._2nd_Shift_Lunch_Length,Lunch_Length) ,MOV(LN00_Weekly_Schedule.Monday.S2_Scheduled,LN00_Schedule.Scheduled_Units) ];
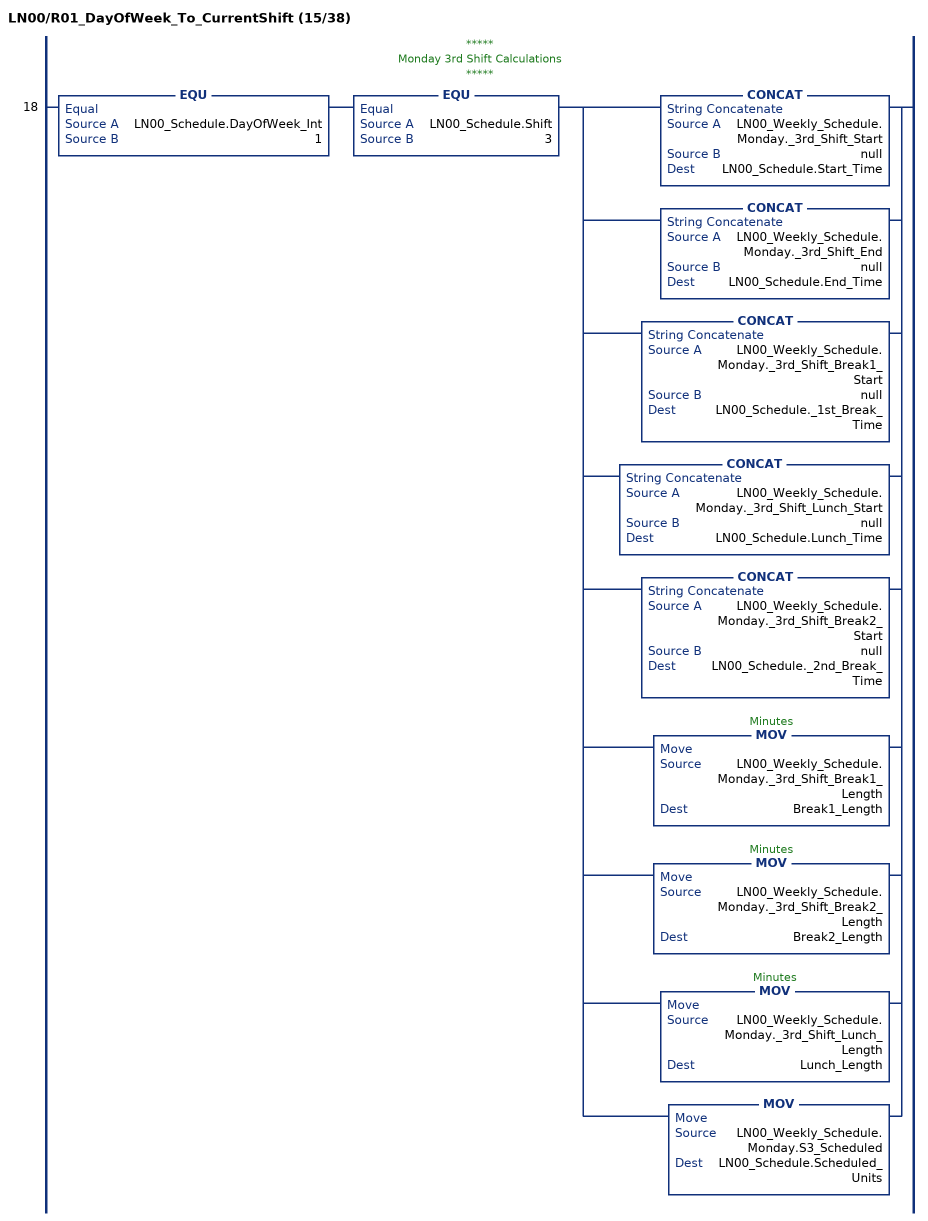
   // *****
   // Monday 3rd Shift Calculations
   // *****
   18: EQU(LN00_Schedule.DayOfWeek_Int,1)EQU(LN00_Schedule.Shift,3)[CONCAT(LN00_Weekly_Schedule.Monday._3rd_Shift_Start,null,LN00_Schedule.Start_Time) ,CONCAT(LN00_Weekly_Schedule.Monday._3rd_Shift_End,null,LN00_Schedule.End_Time) ,CONCAT(LN00_Weekly_Schedule.Monday._3rd_Shift_Break1_Start,null,LN00_Schedule._1st_Break_Time) ,CONCAT(LN00_Weekly_Schedule.Monday._3rd_Shift_Lunch_Start,null,LN00_Schedule.Lunch_Time) ,CONCAT(LN00_Weekly_Schedule.Monday._3rd_Shift_Break2_Start,null,LN00_Schedule._2nd_Break_Time) ,MOV(LN00_Weekly_Schedule.Monday._3rd_Shift_Break1_Length,Break1_Length) ,MOV(LN00_Weekly_Schedule.Monday._3rd_Shift_Break2_Length,Break2_Length) ,MOV(LN00_Weekly_Schedule.Monday._3rd_Shift_Lunch_Length,Lunch_Length) ,MOV(LN00_Weekly_Schedule.Monday.S3_Scheduled,LN00_Schedule.Scheduled_Units) ];
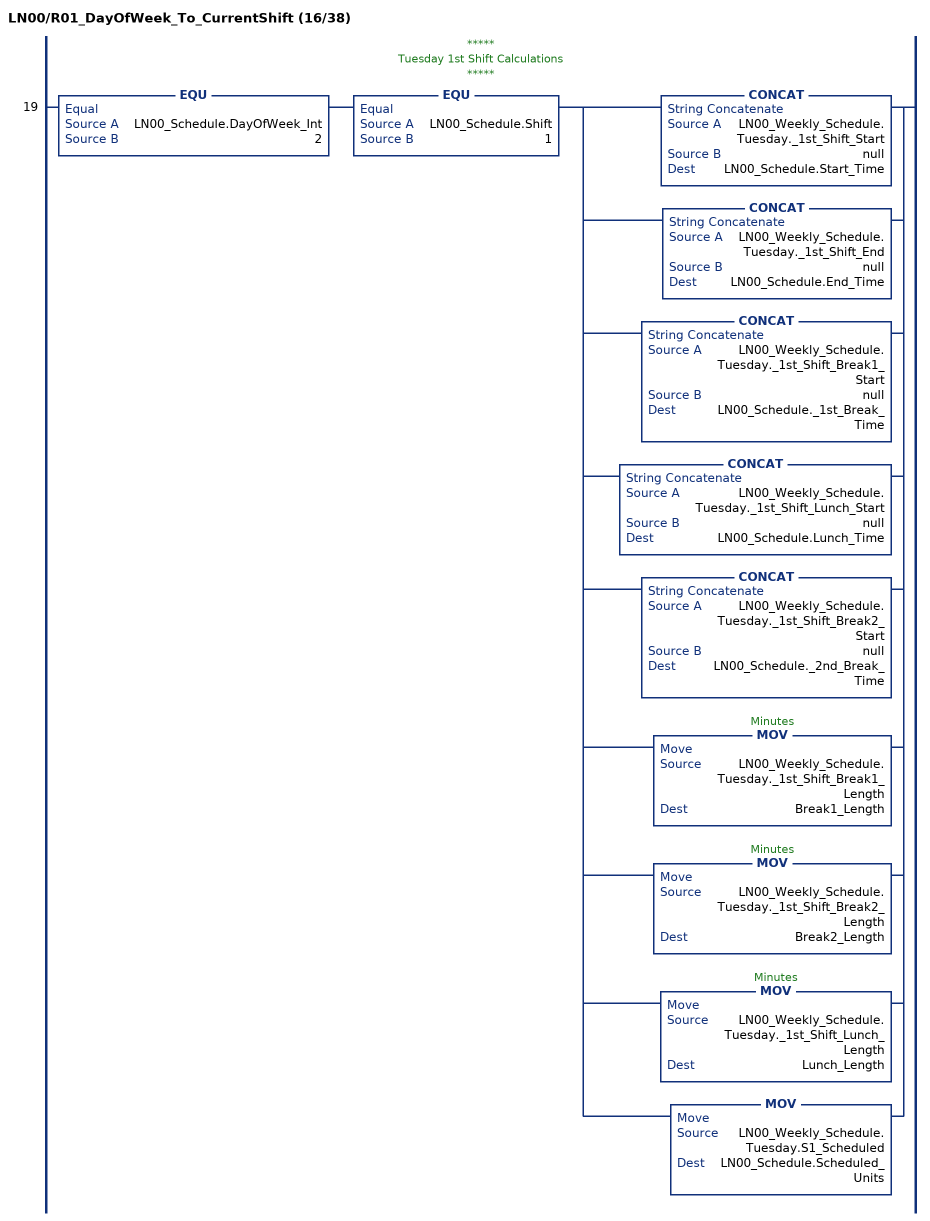
   // *****
   // Tuesday 1st Shift Calculations
   // *****
   19: EQU(LN00_Schedule.DayOfWeek_Int,2)EQU(LN00_Schedule.Shift,1)[CONCAT(LN00_Weekly_Schedule.Tuesday._1st_Shift_Start,null,LN00_Schedule.Start_Time) ,CONCAT(LN00_Weekly_Schedule.Tuesday._1st_Shift_End,null,LN00_Schedule.End_Time) ,CONCAT(LN00_Weekly_Schedule.Tuesday._1st_Shift_Break1_Start,null,LN00_Schedule._1st_Break_Time) ,CONCAT(LN00_Weekly_Schedule.Tuesday._1st_Shift_Lunch_Start,null,LN00_Schedule.Lunch_Time) ,CONCAT(LN00_Weekly_Schedule.Tuesday._1st_Shift_Break2_Start,null,LN00_Schedule._2nd_Break_Time) ,MOV(LN00_Weekly_Schedule.Tuesday._1st_Shift_Break1_Length,Break1_Length) ,MOV(LN00_Weekly_Schedule.Tuesday._1st_Shift_Break2_Length,Break2_Length) ,MOV(LN00_Weekly_Schedule.Tuesday._1st_Shift_Lunch_Length,Lunch_Length) ,MOV(LN00_Weekly_Schedule.Tuesday.S1_Scheduled,LN00_Schedule.Scheduled_Units) ];
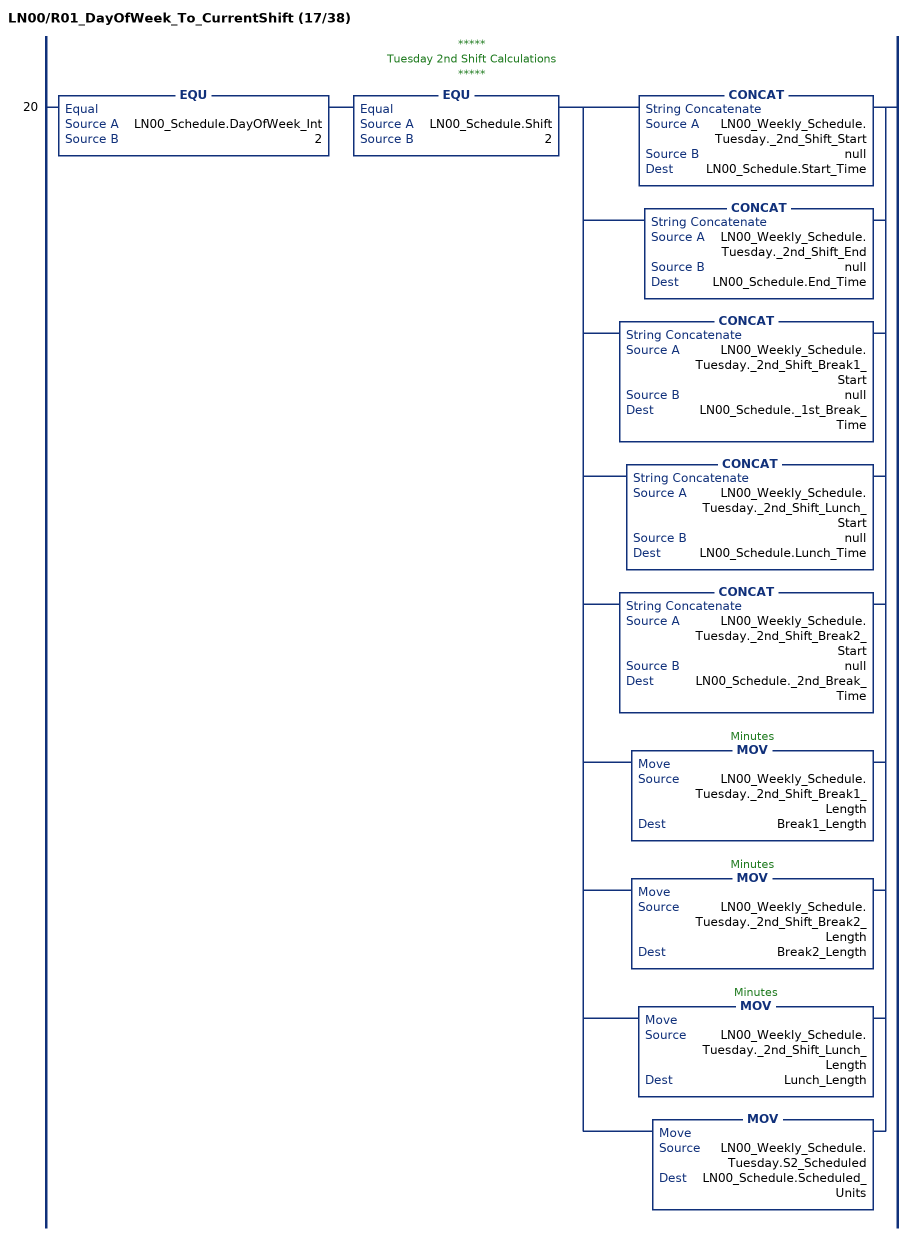
   // *****
   // Tuesday 2nd Shift Calculations
   // *****
   20: EQU(LN00_Schedule.DayOfWeek_Int,2)EQU(LN00_Schedule.Shift,2)[CONCAT(LN00_Weekly_Schedule.Tuesday._2nd_Shift_Start,null,LN00_Schedule.Start_Time) ,CONCAT(LN00_Weekly_Schedule.Tuesday._2nd_Shift_End,null,LN00_Schedule.End_Time) ,CONCAT(LN00_Weekly_Schedule.Tuesday._2nd_Shift_Break1_Start,null,LN00_Schedule._1st_Break_Time) ,CONCAT(LN00_Weekly_Schedule.Tuesday._2nd_Shift_Lunch_Start,null,LN00_Schedule.Lunch_Time) ,CONCAT(LN00_Weekly_Schedule.Tuesday._2nd_Shift_Break2_Start,null,LN00_Schedule._2nd_Break_Time) ,MOV(LN00_Weekly_Schedule.Tuesday._2nd_Shift_Break1_Length,Break1_Length) ,MOV(LN00_Weekly_Schedule.Tuesday._2nd_Shift_Break2_Length,Break2_Length) ,MOV(LN00_Weekly_Schedule.Tuesday._2nd_Shift_Lunch_Length,Lunch_Length) ,MOV(LN00_Weekly_Schedule.Tuesday.S2_Scheduled,LN00_Schedule.Scheduled_Units) ];
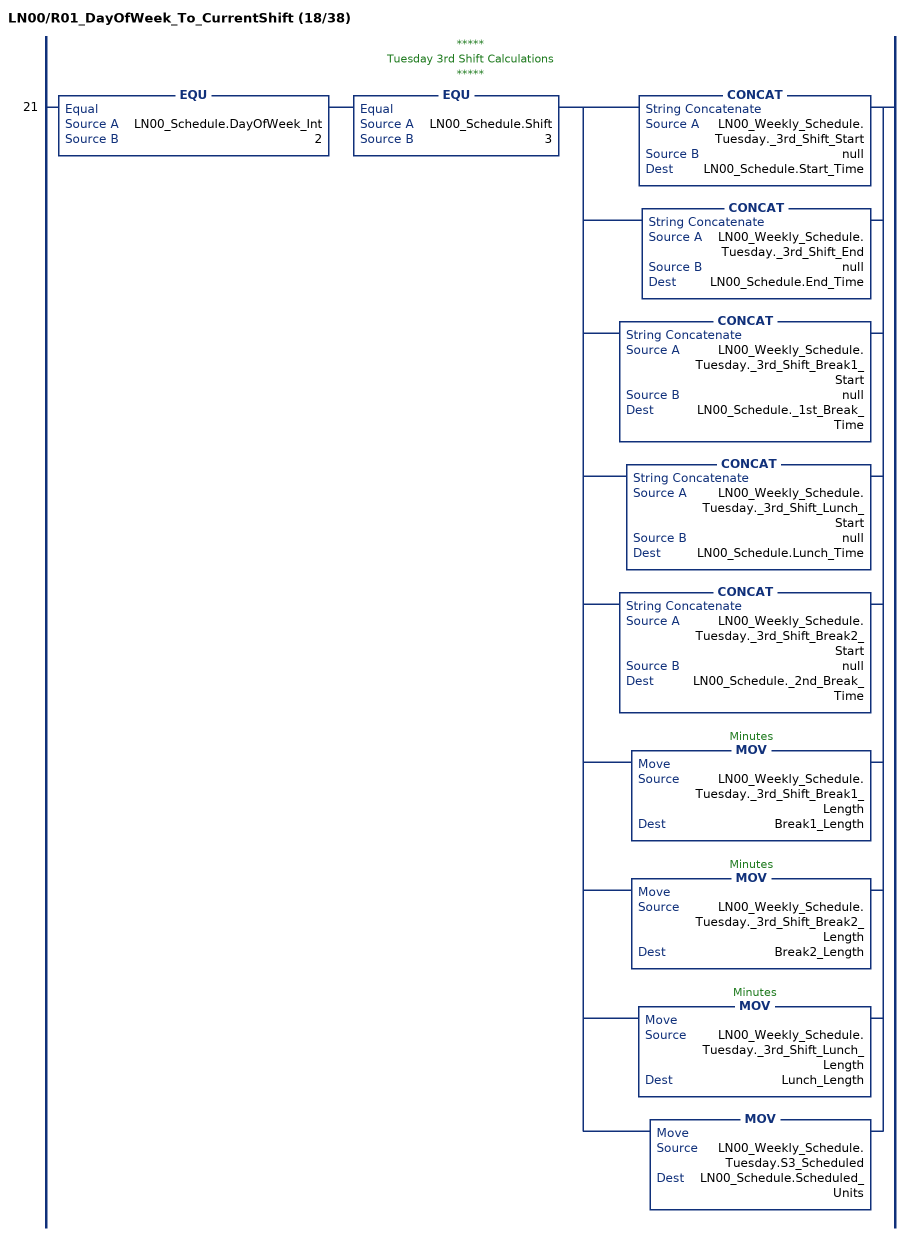
   // *****
   // Tuesday 3rd Shift Calculations
   // *****
   21: EQU(LN00_Schedule.DayOfWeek_Int,2)EQU(LN00_Schedule.Shift,3)[CONCAT(LN00_Weekly_Schedule.Tuesday._3rd_Shift_Start,null,LN00_Schedule.Start_Time) ,CONCAT(LN00_Weekly_Schedule.Tuesday._3rd_Shift_End,null,LN00_Schedule.End_Time) ,CONCAT(LN00_Weekly_Schedule.Tuesday._3rd_Shift_Break1_Start,null,LN00_Schedule._1st_Break_Time) ,CONCAT(LN00_Weekly_Schedule.Tuesday._3rd_Shift_Lunch_Start,null,LN00_Schedule.Lunch_Time) ,CONCAT(LN00_Weekly_Schedule.Tuesday._3rd_Shift_Break2_Start,null,LN00_Schedule._2nd_Break_Time) ,MOV(LN00_Weekly_Schedule.Tuesday._3rd_Shift_Break1_Length,Break1_Length) ,MOV(LN00_Weekly_Schedule.Tuesday._3rd_Shift_Break2_Length,Break2_Length) ,MOV(LN00_Weekly_Schedule.Tuesday._3rd_Shift_Lunch_Length,Lunch_Length) ,MOV(LN00_Weekly_Schedule.Tuesday.S3_Scheduled,LN00_Schedule.Scheduled_Units) ];
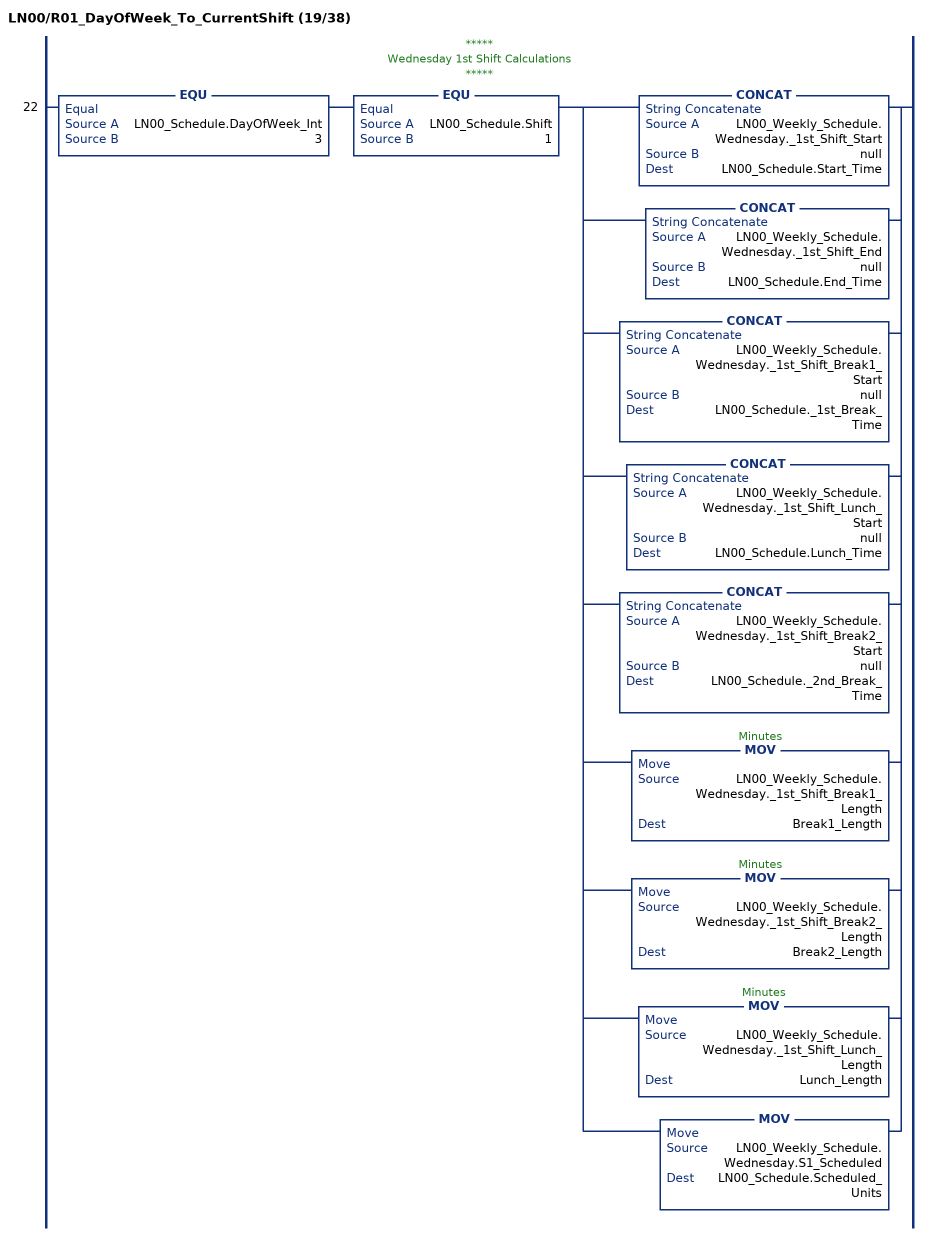
   // *****
   // Wednesday 1st Shift Calculations
   // *****
   22: EQU(LN00_Schedule.DayOfWeek_Int,3)EQU(LN00_Schedule.Shift,1)[CONCAT(LN00_Weekly_Schedule.Wednesday._1st_Shift_Start,null,LN00_Schedule.Start_Time) ,CONCAT(LN00_Weekly_Schedule.Wednesday._1st_Shift_End,null,LN00_Schedule.End_Time) ,CONCAT(LN00_Weekly_Schedule.Wednesday._1st_Shift_Break1_Start,null,LN00_Schedule._1st_Break_Time) ,CONCAT(LN00_Weekly_Schedule.Wednesday._1st_Shift_Lunch_Start,null,LN00_Schedule.Lunch_Time) ,CONCAT(LN00_Weekly_Schedule.Wednesday._1st_Shift_Break2_Start,null,LN00_Schedule._2nd_Break_Time) ,MOV(LN00_Weekly_Schedule.Wednesday._1st_Shift_Break1_Length,Break1_Length) ,MOV(LN00_Weekly_Schedule.Wednesday._1st_Shift_Break2_Length,Break2_Length) ,MOV(LN00_Weekly_Schedule.Wednesday._1st_Shift_Lunch_Length,Lunch_Length) ,MOV(LN00_Weekly_Schedule.Wednesday.S1_Scheduled,LN00_Schedule.Scheduled_Units) ];
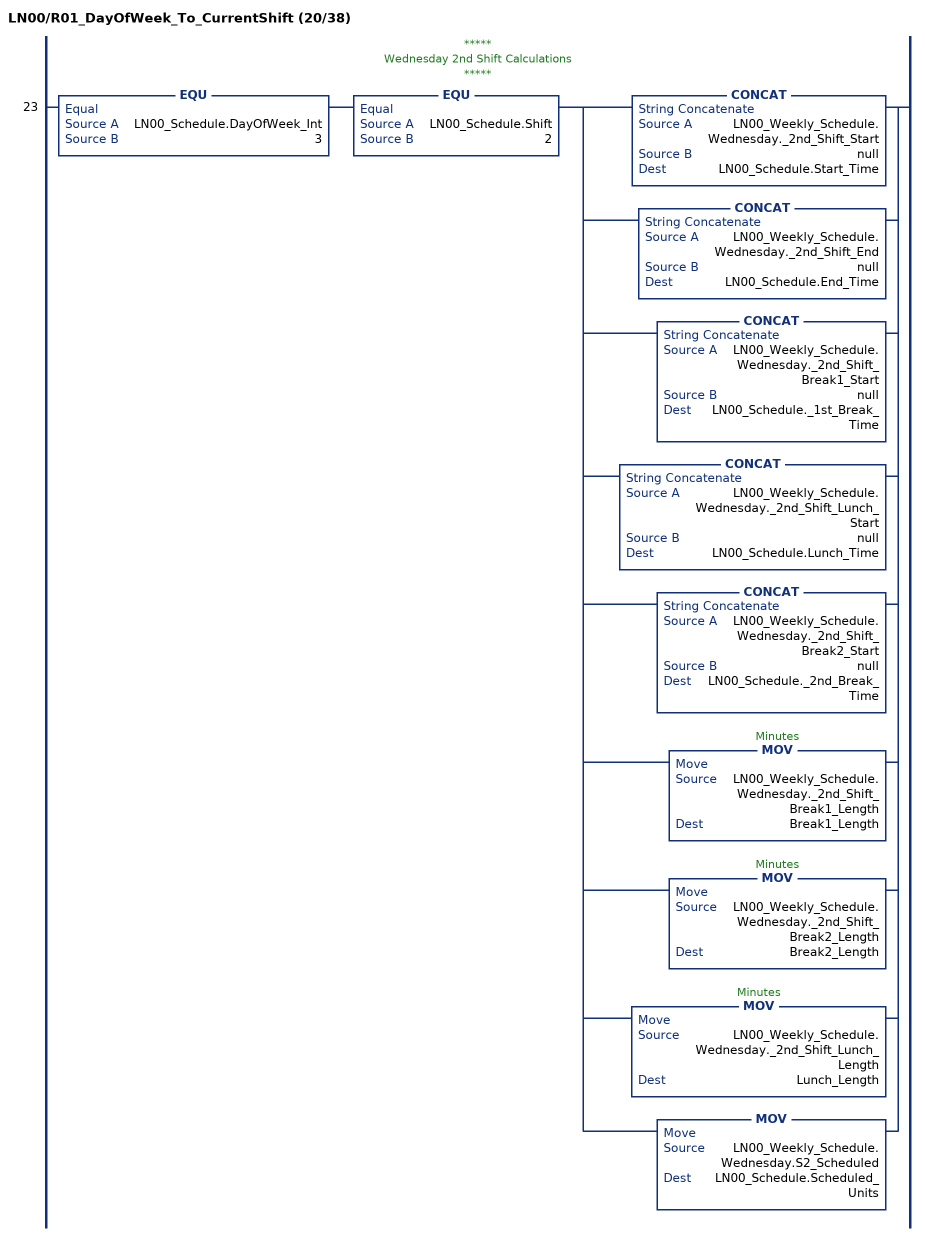
   // *****
   // Wednesday 2nd Shift Calculations
   // *****
   23: EQU(LN00_Schedule.DayOfWeek_Int,3)EQU(LN00_Schedule.Shift,2)[CONCAT(LN00_Weekly_Schedule.Wednesday._2nd_Shift_Start,null,LN00_Schedule.Start_Time) ,CONCAT(LN00_Weekly_Schedule.Wednesday._2nd_Shift_End,null,LN00_Schedule.End_Time) ,CONCAT(LN00_Weekly_Schedule.Wednesday._2nd_Shift_Break1_Start,null,LN00_Schedule._1st_Break_Time) ,CONCAT(LN00_Weekly_Schedule.Wednesday._2nd_Shift_Lunch_Start,null,LN00_Schedule.Lunch_Time) ,CONCAT(LN00_Weekly_Schedule.Wednesday._2nd_Shift_Break2_Start,null,LN00_Schedule._2nd_Break_Time) ,MOV(LN00_Weekly_Schedule.Wednesday._2nd_Shift_Break1_Length,Break1_Length) ,MOV(LN00_Weekly_Schedule.Wednesday._2nd_Shift_Break2_Length,Break2_Length) ,MOV(LN00_Weekly_Schedule.Wednesday._2nd_Shift_Lunch_Length,Lunch_Length) ,MOV(LN00_Weekly_Schedule.Wednesday.S2_Scheduled,LN00_Schedule.Scheduled_Units) ];
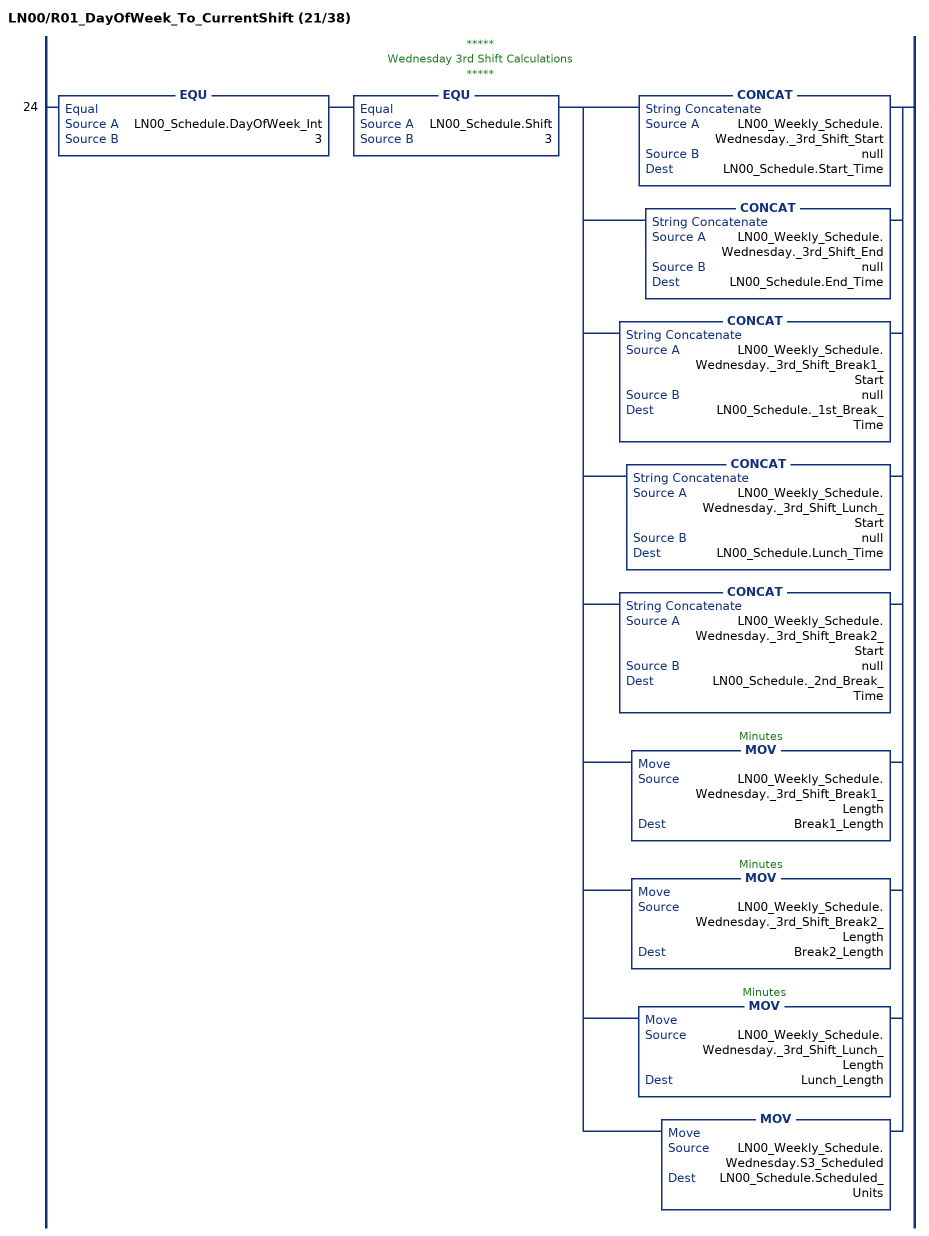
   // *****
   // Wednesday 3rd Shift Calculations
   // *****
   24: EQU(LN00_Schedule.DayOfWeek_Int,3)EQU(LN00_Schedule.Shift,3)[CONCAT(LN00_Weekly_Schedule.Wednesday._3rd_Shift_Start,null,LN00_Schedule.Start_Time) ,CONCAT(LN00_Weekly_Schedule.Wednesday._3rd_Shift_End,null,LN00_Schedule.End_Time) ,CONCAT(LN00_Weekly_Schedule.Wednesday._3rd_Shift_Break1_Start,null,LN00_Schedule._1st_Break_Time) ,CONCAT(LN00_Weekly_Schedule.Wednesday._3rd_Shift_Lunch_Start,null,LN00_Schedule.Lunch_Time) ,CONCAT(LN00_Weekly_Schedule.Wednesday._3rd_Shift_Break2_Start,null,LN00_Schedule._2nd_Break_Time) ,MOV(LN00_Weekly_Schedule.Wednesday._3rd_Shift_Break1_Length,Break1_Length) ,MOV(LN00_Weekly_Schedule.Wednesday._3rd_Shift_Break2_Length,Break2_Length) ,MOV(LN00_Weekly_Schedule.Wednesday._3rd_Shift_Lunch_Length,Lunch_Length) ,MOV(LN00_Weekly_Schedule.Wednesday.S3_Scheduled,LN00_Schedule.Scheduled_Units) ];
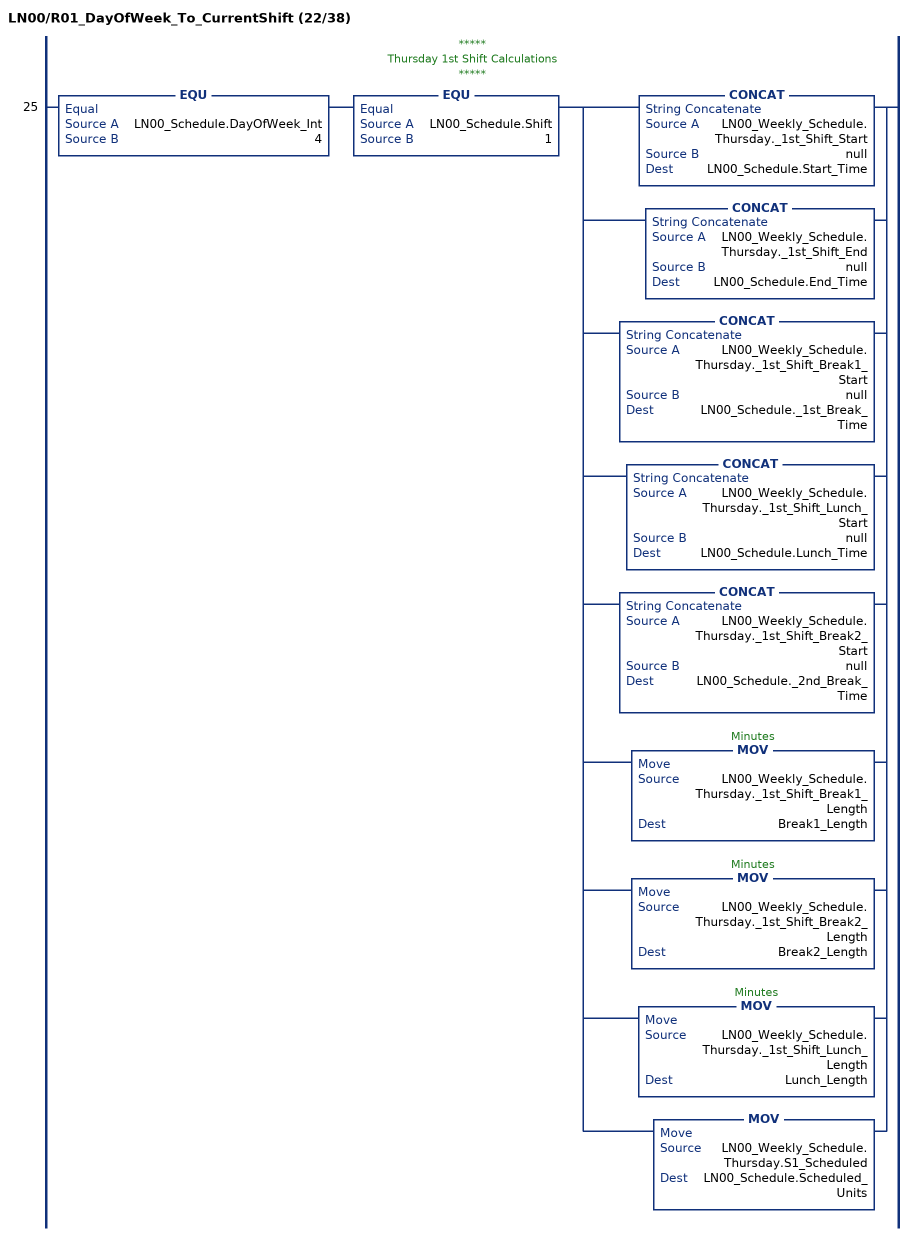
   // *****
   // Thursday 1st Shift Calculations
   // *****
   25: EQU(LN00_Schedule.DayOfWeek_Int,4)EQU(LN00_Schedule.Shift,1)[CONCAT(LN00_Weekly_Schedule.Thursday._1st_Shift_Start,null,LN00_Schedule.Start_Time) ,CONCAT(LN00_Weekly_Schedule.Thursday._1st_Shift_End,null,LN00_Schedule.End_Time) ,CONCAT(LN00_Weekly_Schedule.Thursday._1st_Shift_Break1_Start,null,LN00_Schedule._1st_Break_Time) ,CONCAT(LN00_Weekly_Schedule.Thursday._1st_Shift_Lunch_Start,null,LN00_Schedule.Lunch_Time) ,CONCAT(LN00_Weekly_Schedule.Thursday._1st_Shift_Break2_Start,null,LN00_Schedule._2nd_Break_Time) ,MOV(LN00_Weekly_Schedule.Thursday._1st_Shift_Break1_Length,Break1_Length) ,MOV(LN00_Weekly_Schedule.Thursday._1st_Shift_Break2_Length,Break2_Length) ,MOV(LN00_Weekly_Schedule.Thursday._1st_Shift_Lunch_Length,Lunch_Length) ,MOV(LN00_Weekly_Schedule.Thursday.S1_Scheduled,LN00_Schedule.Scheduled_Units) ];
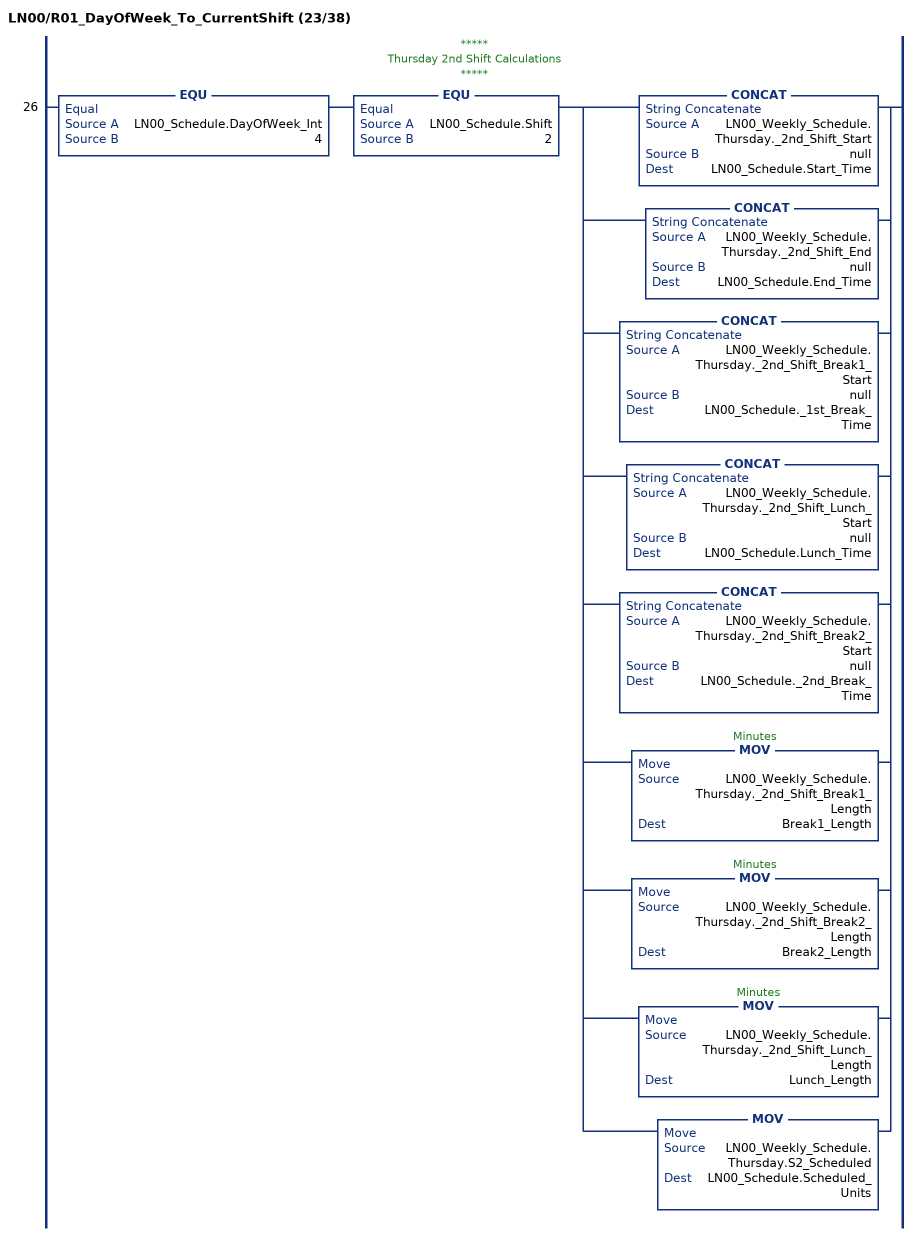
   // *****
   // Thursday 2nd Shift Calculations
   // *****
   26: EQU(LN00_Schedule.DayOfWeek_Int,4)EQU(LN00_Schedule.Shift,2)[CONCAT(LN00_Weekly_Schedule.Thursday._2nd_Shift_Start,null,LN00_Schedule.Start_Time) ,CONCAT(LN00_Weekly_Schedule.Thursday._2nd_Shift_End,null,LN00_Schedule.End_Time) ,CONCAT(LN00_Weekly_Schedule.Thursday._2nd_Shift_Break1_Start,null,LN00_Schedule._1st_Break_Time) ,CONCAT(LN00_Weekly_Schedule.Thursday._2nd_Shift_Lunch_Start,null,LN00_Schedule.Lunch_Time) ,CONCAT(LN00_Weekly_Schedule.Thursday._2nd_Shift_Break2_Start,null,LN00_Schedule._2nd_Break_Time) ,MOV(LN00_Weekly_Schedule.Thursday._2nd_Shift_Break1_Length,Break1_Length) ,MOV(LN00_Weekly_Schedule.Thursday._2nd_Shift_Break2_Length,Break2_Length) ,MOV(LN00_Weekly_Schedule.Thursday._2nd_Shift_Lunch_Length,Lunch_Length) ,MOV(LN00_Weekly_Schedule.Thursday.S2_Scheduled,LN00_Schedule.Scheduled_Units) ];
